END_CASE
///============================================================================================}}}
///(*==================================== Sorting station ====================================*){{{
(* Add buffer for sorting station *)
CASE eFinalResult OF
	VISION_RESULT_UNKNOWN:
		;
	VISION_RESULT_GOOD:
		Buffer_SortGood.A_Add(in := fbRotaryTable.ActualPosition + lrSortGoodDistance);
		eFinalResult 		:= VISION_RESULT_UNKNOWN;
	VISION_RESULT_CONTAMINATION_DIRTY:
		Buffer_SortDirt.A_Add(in := fbRotaryTable.ActualPosition + lrSortDirtDistance);
		eFinalResult 		:= VISION_RESULT_UNKNOWN;
	VISION_RESULT_SCRATCH_DENT:
		Buffer_SortDent.A_Add(in := fbRotaryTable.ActualPosition + lrSortDentDistance);
		eFinalResult 		:= VISION_RESULT_UNKNOWN;
	VISION_RESULT_REJECT:
		Buffer_SortReject.A_Add(in := fbRotaryTable.ActualPosition + lrSortRejectDistance);
		eFinalResult 		:= VISION_RESULT_UNKNOWN;

END_CASE
(* Shoot the product out *)
(* Good case *)
CASE uSortGoodGetPosState OF
	0://idle | check buffer
		IF Buffer_SortGood.nCount > 0 THEN
			uSortGoodGetPosState:= 10;
		END_IF
	10://get position
		Buffer_SortGood.A_Get(out => lrSortGoodPos);
		uSortGoodGetPosState := 20;
	20://waiting table move in position | command table
		bResultProcessing 	:= FALSE;
		IF LREAL_TO_INT(fbRotaryTable.ActualPosition) <= LREAL_TO_INT(lrSortGoodPos) THEN
			uSortGoodGetPosState := 30;
		END_IF
	30://shoot it
		Buffer_SortGood.A_Remove(out => lrSortGoodPos);
		doBlowGood.Out := TRUE;
		uSortGoodGetPosState := 40;
		
	40://off
		tonGoodDelay(IN := TRUE, PT := tSortValveGoodTime);
		IF tonGoodDelay.Q THEN	
			doBlowGood.Out := FALSE;
			tonGoodDelay.IN := FALSE;
			uSortGoodGetPosState := 0;
		END_IF
		
END_CASE
(* DIRT CASE *)
CASE uSortDirtGetPosState OF
	0://idle | check buffer
		IF Buffer_SortDirt.nCount > 0 THEN
			uSortDirtGetPosState:= 10;
		END_IF
	10://get position
		Buffer_SortDirt.A_Get(out => lrSortDirtPos);
		uSortDirtGetPosState := 20;
	20://waiting table move in position | command table
		bResultProcessing 	:= FALSE;
		IF LREAL_TO_INT(fbRotaryTable.ActualPosition) <= LREAL_TO_INT(lrSortDirtPos) THEN
			uSortDirtGetPosState := 30;
		END_IF
	30://shoot it
		Buffer_SortDirt.A_Remove(out => lrSortDirtPos);
		doBlowDirtScratch.Out := TRUE;
		uSortDirtGetPosState := 40;
		
	40://off
		tonDirtDelay(IN := TRUE, PT := tSortValveDirtTime);
		IF tonDirtDelay.Q THEN	
			doBlowDirtScratch.Out := FALSE;
			tonDirtDelay.IN := FALSE;
			uSortDirtGetPosState := 0;
		END_IF
		
END_CASE
(* DENT CASE *)
CASE uSortDentGetPosState OF
	0://idle | check buffer
		IF Buffer_SortDent.nCount > 0 THEN
			uSortDentGetPosState:= 10;
		END_IF
	10://get position
		Buffer_SortDent.A_Get(out => lrSortDentPos);
		uSortDentGetPosState := 20;
	20://waiting table move in position | command table
		bResultProcessing 	:= FALSE;
		IF LREAL_TO_INT(fbRotaryTable.ActualPosition) <= LREAL_TO_INT(lrSortDentPos) THEN
			uSortDentGetPosState := 30;
		END_IF
	30://shoot it
		Buffer_SortDent.A_Remove(out => lrSortDentPos);
		doBlowDentContamination.Out := TRUE;
		uSortDentGetPosState := 40;
		
	40://off
		tonDentDelay(IN := TRUE, PT := tSortValveDentTime);
		IF tonDentDelay.Q THEN	
			doBlowDentContamination.Out := FALSE;
			tonDentDelay.IN := FALSE;
			uSortDentGetPosState := 0;
		END_IF
		
END_CASE
(* REJECT CASE *)
CASE uSortRejectGetPosState OF
	0://idle | check buffer
		IF Buffer_SortReject.nCount > 0 THEN
			uSortRejectGetPosState:= 10;
		END_IF
	10://get position
		Buffer_SortReject.A_Get(out => lrSortRejectPos);
		uSortRejectGetPosState := 20;
	20://waiting table move in position | command table
		bResultProcessing 	:= FALSE;
		IF LREAL_TO_INT(fbRotaryTable.ActualPosition) <= LREAL_TO_INT(lrSortRejectPos) THEN
			uSortRejectGetPosState := 30;
		END_IF
	30://shoot it
		Buffer_SortReject.A_Remove(out => lrSortRejectPos);
		doBlowReject.Out := TRUE;
		uSortRejectGetPosState := 40;
		
	40://off
		tonRejectDelay(IN := TRUE, PT := tSortValveRejectTime);
		IF tonRejectDelay.Q THEN	
			doBlowReject.Out := FALSE;
			tonRejectDelay.IN := FALSE;
			uSortRejectGetPosState := 0;
		END_IF
		
END_CASE
///============================================================================================}}}
(* control param *)
fbRobot.ref_CR800.Override:= 5;
uBufferTableCount:= Buffer_RotaryTable.nCount;

(* Mornitoring param *)
bActive 			:= fbRotaryTable.Active;
bBusy				:= fbRotaryTable.Busy;
bError 				:= fbRotaryTable.Error;
iErrorID 			:= fbRotaryTable.ErrorID;
iAxisErrorID 		:= fbRotaryTable.ErrorID;
lrActualPosition 	:= fbRotaryTable.ActualPosition;
rActualVelocity		:= fbRotaryTable.ActualVelocity;
bPowerOn 			:= fbRotaryTable.PowerOn;
bIsHomed 			:= fbRotaryTable.IsHomed;
bInVelocity			:= fbRotaryTable.InVelocity;
bInPostion 			:= fbRotaryTable.InPosition;
bMoveActive 		:= fbRotaryTable.MoveActive;
bJogDone 			:= fbRotaryTable.JogDone;
bStopped 			:= fbRotaryTable.Stopped;
bHalted 			:= fbRotaryTable.Halted;
eStatePlcOpen		:= fbRotaryTable.StatePlcOpen;

fbRobot.ref_CR800.Override:= 30;
fbRotaryTable.Velocity 			:= 50.0;
END_METHOD

METHOD PROTECTED Production_fixing : BOOL
VAR_INST
	(* Robot *)
	RobotState 					: UINT;
	
	(* Table *)
	TableState					: UINT;
	OneStep 					: LREAL:= -30.0; //-61.1928;	(* Define by the distance between station 3 and 4 *)
	lrRelativeDistance 			: LREAL;
	bProductAboveTable 			: BOOL;				(* Signal Robot is at the table *)
	bGetPictureStation3			: BOOL; 			(* Cmd get picture st3 to vision system *)
	bGetPictureStation4 		: BOOL; 			(* Cmd get picture st4 to vision system *)
	bResultProcessing 			: BOOL;				(* Request result from vision system, then add buffer for sorting station *)
	
	(* Buffer *)
	BufferState : UINT;
	Buffer_RotaryTable			: FB_DataSetFifo_1; 	(* Contain the position of all product on the table *)
	Buffer_Station3				: FB_DataSetFifo_1;	(* Contain the trigger position *)
	Buffer_Station4				: FB_DataSetFifo_1;	(* Contain the trigger position *)
	
	(* Sorting Station *)
	Buffer_SortGood				: FB_DataSetFifo_1;
	Buffer_SortDirt				: FB_DataSetFifo_1;
	Buffer_SortDent				: FB_DataSetFifo_1;
	Buffer_SortReject			: FB_DataSetFifo_1;
	
	
	
	lrSortGoodPos				: LREAL;
	lrSortDirtPos				: LREAL;
	lrSortDentPos				: LREAL;
	lrSortRejectPos				: LREAL;
	
	uSortGoodGetPosState		: UINT; 			(* state machine of get sort position from buffer *)
	uSortDirtGetPosState		: UINT;
	uSortDentGetPosState		: UINT;
	uSortRejectGetPosState		: UINT;
		
	tonGoodDelay				: TON;				(* one shoot of good delay valve *)
	tonDirtDelay				: TON;				(* one shoot of dirt delay valve *)
	tonDentDelay				: TON;				(* one shoot of dent delay valve *)								
	tonRejectDelay				: TON;				(* one shoot of reject delay valve *)	
							

	
	(*=== Vision ===*)
	Vision3State 		: UINT;
	Vision4State		: UINT;
	lrCapPosStation3 	: LREAL;
	lrCapPosStation4	: LREAL;
	bGood 				: BOOL;
	bAtVision3 			: BOOL;	(* Product is at vision 3 *)
	bAtVision4 			: BOOL;	(* Product is at vision 4 *)
	eFinalResult		: E_VisionResult;

	(* Axis status flags *)
	bActive					: BOOL;
	bBusy					: BOOL;								(* Function block currently executes one of the requests *)
	bError					: BOOL;								(* Error status flag *)
	iErrorID				: UDINT;							(* Error ID *)
	iAxisErrorID			: UDINT;							(* Axis error ID*)
	lrActualPosition		: LREAL;							(* Actual axis position in selected units *)
	rActualVelocity			: REAL;								(* Actual axis velocity in selected units *)
	bPowerOn 				: BOOL;								(* Power On status bit *)
	bIsHomed				: BOOL;								(* Axis has been homed even once *)
	bInVelocity				: BOOL;								(* Axis is moving in target velocity *)
	bInPostion				: BOOL;								(* Axis reached target position *)
	bMoveActive				: BOOL;								(* Axis is moving to target position *)
	bJogDone				: BOOL;								(* Axis manual movement by jog done *)
	bStopped				: BOOL;								(* Axis movement has been stopped *)
	bHalted					: BOOL;								(* Axis movement has been halted *)
	eStatePlcOpen			: E_AxisStatePlcOpen;
	
	uBufferTableCount : UDINT;
	
	(* testing bit *)
	bResultTest : BOOL;
	bResultGood : BOOL;
	bResultDirt : BOOL;
	bResultDent : BOOL;
	bResultReject : BOOL;

	(**)
	iTableSupervisor 	: UINT;
	iTableExecutor 		: UINT;
	
	Buffer_Sorting		: FB_DataSetFifo_1;	(* Contain the trigger position *)
	
	lrStation3Location : LREAL;
	lrStation4Location : LREAL;
	lrStationSortLocation : LREAL;
	lrTargetLocation : LREAL;
	
	bBufferTest : BOOL;
	
END_VAR
///(*==================================== Robot + Vision process ====================================*){{{
CASE RobotState OF	
	0://IDLE go bowl
		fbRobot.MR_GoBowl();
		IF NOT fbRobot.Busy THEN
			RobotState := 5;
		END_IF		
	5://product detected
		IF diProductPresenceBowl.In THEN (* waiting product *)
			RobotState := 6;
		END_IF
	
	6://go input
		fbRobot.MR_GoInputProduct();
		IF NOT fbRobot.Busy THEN
			RobotState := 7;
		END_IF
		
	7://robot pick
		fbRobot.MR_Pick();
		IF NOT fbRobot.Busy THEN
			RobotState := 10;
		END_IF 
		
	10://go to station 1
		fbRobot.MR_GoStation1();
		IF NOT fbRobot.Busy THEN
			RobotState := 20;
		END_IF
		
	20://double trig cam 1+2
		IF doTriggerCam1.Command(PulseWidth:=T#1MS, DelayTimeForSecondTrigger := T#35MS) AND
			doTriggerCam2.Command(PulseWidth:=T#1MS, DelayTimeForSecondTrigger := T#35MS) THEN
			RobotState:= 30;
		END_IF
	30://go to station 2
		fbRobot.MR_GoStation2();
		IF NOT fbRobot.Busy THEN
			RobotState := 40;
		END_IF
	40://double trig cam 3+4
		IF doTriggerCam3.Command(PulseWidth:=T#1MS, DelayTimeForSecondTrigger := T#35MS) AND
			doTriggerCam4.Command(PulseWidth:=T#1MS, DelayTimeForSecondTrigger := T#35MS) THEN
			RobotState := 50;
		END_IF
	50://goto rotary table
		fbRobot.MR_GoRotaryTable();
		IF NOT fbRobot.Busy THEN
			bProductAboveTable := TRUE;		
			RobotState:= 60;
		END_IF
	60://waiting command from table
		;
		
END_CASE
///============================================================================================}}}
(* TABLE SUPERVISOR *)
CASE iTableSupervisor OF
	0:
		IF bProductAboveTable THEN			
			IF iTableExecutor = 0 THEN//IDLE
				RobotState:=60;
			END_IF
		END_IF
		
END_CASE
(* TABLE EXECUTOR *)
CASE iTableExecutor OF
	0: //IDLE
		;
	10://TAKE PRODUCT
		
	20://ADD BUFFER
		Buffer_Station3.A_Add(in:= fbRotaryTable.ActualPosition + 2*OneStep); 	(* station position *)
		Buffer_Station4.A_Add(in:= fbRotaryTable.ActualPosition + 4*OneStep);	(* station position *)
		
		Buffer_RotaryTable.A_Add(in:= fbRotaryTable.ActualPosition + OneStep);	(* place position *)
		Buffer_RotaryTable.A_Add(in:= fbRotaryTable.ActualPosition + OneStep);	(* place position *)
		Buffer_RotaryTable.A_Add(in:= fbRotaryTable.ActualPosition + OneStep);	(* place position *)
		Buffer_RotaryTable.A_Add(in:= fbRotaryTable.ActualPosition + OneStep);	(* place position *)
		
		iTableExecutor := 30;
	30://calc the position
		IF Buffer_Station3.nCount > 0 AND Buffer_Station4.nCount > 0 THEN
			Buffer_Station3.A_Get(out => lrStation3Location);
			Buffer_Station4.A_Get(out => lrStation4Location);
			
			IF LREAL_TO_LINT(lrStation3Location) > LREAL_TO_LINT(lrStation4Location) THEN
				lrTargetLocation := lrStation3Location;
				Buffer_Station3.A_Remove(out => lrStation3Location);
				
			ELSIF LREAL_TO_LINT(lrStation3Location) < LREAL_TO_LINT(lrStation4Location) THEN
				lrTargetLocation := lrStation4Location;
				Buffer_Station4.A_Remove(out => lrStation4Location);
				
			ELSE
				lrTargetLocation := lrStation3Location;
				Buffer_Station3.A_Remove(out => lrStation3Location);
				Buffer_Station4.A_Remove(out => lrStation4Location);
			
			END_IF
			iTableExecutor := 40;
			
		ELSIF Buffer_Station3.nCount = 0 AND Buffer_Station4.nCount = 0 THEN
			iTableExecutor := 0;//IDLE
			
		ELSE
			IF Buffer_Station3.nCount = 0 THEN
				lrTargetLocation := lrStation4Location;
				Buffer_Station4.A_Remove(out => lrStation4Location);
				
			ELSE
				lrTargetLocation := lrStation3Location;
				Buffer_Station3.A_Remove(out => lrStation3Location);
				
			END_IF
			iTableExecutor := 40;
		END_IF
		
	40://
		fbRotaryTable.MR_MoveAbsolute(lrAbsolutePosition := lrTargetLocation);
		IF fbRotaryTable.InPosition THEN
			iTableExecutor := 30;
		END_IF
		
		
END_CASE
///============================================================================================}}}
(* control param *)
fbRobot.ref_CR800.Override:= 5;
uBufferTableCount:= Buffer_RotaryTable.nCount;

(* Mornitoring param *)
bActive 			:= fbRotaryTable.Active;
bBusy				:= fbRotaryTable.Busy;
bError 				:= fbRotaryTable.Error;
iErrorID 			:= fbRotaryTable.ErrorID;
iAxisErrorID 		:= fbRotaryTable.ErrorID;
lrActualPosition 	:= fbRotaryTable.ActualPosition;
rActualVelocity		:= fbRotaryTable.ActualVelocity;
bPowerOn 			:= fbRotaryTable.PowerOn;
bIsHomed 			:= fbRotaryTable.IsHomed;
bInVelocity			:= fbRotaryTable.InVelocity;
bInPostion 			:= fbRotaryTable.InPosition;
bMoveActive 		:= fbRotaryTable.MoveActive;
bJogDone 			:= fbRotaryTable.JogDone;
bStopped 			:= fbRotaryTable.Stopped;
bHalted 			:= fbRotaryTable.Halted;
eStatePlcOpen		:= fbRotaryTable.StatePlcOpen;

fbRobot.ref_CR800.Override:= 30;
fbRotaryTable.Velocity 			:= 50.0;
END_METHOD

METHOD PROTECTED Robot_Process
VAR_INST
	(* Equipment module sequences *)
	RobotState : UINT;
	
END_VAR
CASE RobotState OF	
	0://IDLE go bowl
		fbRobot.MR_GoBowl();
		IF NOT fbRobot.Busy THEN
			RobotState := 5;
		END_IF		
	5://product detected
		IF diProductPresenceBowl.In THEN (* waiting product *)
			RobotState := 6;
		END_IF
	
	6://go input
		fbRobot.MR_GoInputProduct();
		IF NOT fbRobot.Busy THEN
			RobotState := 7;
		END_IF
		
	7://robot pick
		fbRobot.MR_Pick();
		IF NOT fbRobot.Busy THEN
			RobotState := 10;
		END_IF 
		
	10://go to station 1
		fbRobot.MR_GoStation1();
		IF NOT fbRobot.Busy THEN
			RobotState := 20;
		END_IF
		
	20://double trig cam 1+2
		IF doTriggerCam1.Command(PulseWidth:=T#1MS, DelayTimeForSecondTrigger := T#35MS) AND
			doTriggerCam2.Command(PulseWidth:=T#1MS, DelayTimeForSecondTrigger := T#35MS) THEN
			RobotState:= 30;
		END_IF
	30://go to station 2
		fbRobot.MR_GoStation2();
		IF NOT fbRobot.Busy THEN
			RobotState := 40;
		END_IF
	40://double trig cam 3+4
		IF doTriggerCam3.Command(PulseWidth:=T#1MS, DelayTimeForSecondTrigger := T#35MS) AND
			doTriggerCam4.Command(PulseWidth:=T#1MS, DelayTimeForSecondTrigger := T#35MS) THEN
			RobotState := 50;
		END_IF
	50://goto rotary table
		fbRobot.MR_GoRotaryTable();
		IF NOT fbRobot.Busy THEN
			//bProductAboveTable := TRUE;		
			RobotState:= 60;
		END_IF
	60://waiting command from table
		fbRobot.MR_Place();
		IF NOT fbRobot.Busy THEN
			RobotState := 0;
		END_IF
		
END_CASE
END_METHOD

METHOD robotcamtest : BOOL
VAR_INST
	RobotProcess:UINT;
END_VAR
fbRobot.ref_CR800.Override:= 5;
CASE RobotProcess OF
	
	0://IDLE go bowl
		fbRobot.MR_GoBowl();
		IF NOT fbRobot.Busy THEN
			RobotProcess := 5;
		END_IF		
	5://product detected
		IF diProductPresenceBowl.In THEN (* waiting product *)
			RobotProcess := 6;
		END_IF
	
	6://go input
		fbRobot.MR_GoInputProduct();
		IF NOT fbRobot.Busy THEN
			RobotProcess := 7;
		END_IF
		
	7://robot pick
		fbRobot.MR_Pick();
		IF NOT fbRobot.Busy THEN
			RobotProcess := 10;
		END_IF 
		
	10://go to station 1
		fbRobot.MR_GoStation1();
		IF NOT fbRobot.Busy THEN
			RobotProcess := 20;
		END_IF
END_CASE
END_METHOD

PROPERTY Robots : REFERENCE TO FB_Robot
GET
Robots REF= fbRobot;
END_GET
END_PROPERTY

PROPERTY StateInit : REFERENCE TO E_MachineCtrlStateInit
GET
StateInit REF= eMachineStateInit;
END_GET
END_PROPERTY

PROPERTY StateUninitialized : REFERENCE TO E_MachineCtrlStateUninitialized
GET
StateUninitialized REF= eMachineStateUninitialized;
END_GET
END_PROPERTY

METHOD TableProcess : BOOL
VAR_INST
	(*=== Table ===*)
	TableState : UINT;
	OneStep : LREAL:= -61.1928;
	lrRelativeDistance : LREAL;
	
	(* Axis status flags *)
	bActive					: BOOL;
	bBusy					: BOOL;								(* Function block currently executes one of the requests *)
	bError					: BOOL;								(* Error status flag *)
	iErrorID				: UDINT;							(* Error ID *)
	iAxisErrorID			: UDINT;							(* Axis error ID*)
	lrActualPosition		: LREAL;							(* Actual axis position in selected units *)
	rActualVelocity			: REAL;								(* Actual axis velocity in selected units *)
	bPowerOn 				: BOOL;								(* Power On status bit *)
	bIsHomed				: BOOL;								(* Axis has been homed even once *)
	bInVelocity				: BOOL;								(* Axis is moving in target velocity *)
	bInPostion				: BOOL;								(* Axis reached target position *)
	bMoveActive				: BOOL;								(* Axis is moving to target position *)
	bJogDone				: BOOL;								(* Axis manual movement by jog done *)
	bStopped				: BOOL;								(* Axis movement has been stopped *)
	bHalted					: BOOL;								(* Axis movement has been halted *)
	eStatePlcOpen			: E_AxisStatePlcOpen;				(* Current PLCOpen state of axis *)
	
	
	(* Buffer *)
	Buffer_RotaryTable			: FB_DataSetFifo; 	(* Contain the position of all product on the table *)
	Buffer_Station3				: FB_DataSetFifo;	(* Contain the trigger position *)
	Buffer_Station4				: FB_DataSetFifo;	(* Contain the trigger position *)
	
	(*=== Vision ===*)
	Vision3State : UINT;
	Vision4State: UINT;
	lrCapPosStation3 : LREAL;
	lrCapPosStation4: LREAL;
	//lrActualPosition :LREAL;
	bBufferReset : BOOL;
END_VAR
CASE TableState OF
	0://product in
		IF diProductPresenceBowl.In THEN (* waiting product *)
			TableState := 10;
		END_IF
	10://buffer table, station 3, station 4
		IF Buffer_RotaryTable.Add2Data(in1 := OneStep, in2 := OneStep) THEN
			IF Buffer_Station3.Add1Data(in := fbRotaryTable.ActualPosition + OneStep) THEN
				IF Buffer_Station4.Add1Data(in := fbRotaryTable.ActualPosition + 2*OneStep) THEN
					TableState := 20;
		
				END_IF				
			END_IF
		END_IF
	20://take distance
		Buffer_RotaryTable.Remove(out => lrRelativeDistance);
		IF Buffer_RotaryTable.OK THEN
			TableState := 30;
		END_IF
	30://move distance
		fbRotaryTable.MR_MoveRelative(lrRelativeDistance);
		IF fbRotaryTable.InPosition THEN
			TableState := 40;
		END_IF
	40://check
		IF Buffer_RotaryTable.Count >0 THEN
			TableState := 20;
		ELSE 
			TableState := 0;
		END_IF
END_CASE

lrActualPosition := fbRotaryTable.ActualPosition;

CASE Vision3State OF
	0://take capture position
		Buffer_Station3.Remove(out => lrCapPosStation3);
		IF Buffer_Station3.OK THEN
			Vision3State := 10;
		END_IF
	10://waiting table move in pos
		IF LREAL_TO_INT(fbRotaryTable.ActualPosition) = LREAL_TO_INT(lrCapPosStation3) THEN
			Vision3State:= 20;
			
		END_IF
	20://capture
		IF fbRTCVision.M_CommandStation3(PulseWidth:= T#1MS, DelayTimeForSecondTrigger:= T#33MS) THEN
			Vision3State:= 0;
		END_IF

END_CASE

CASE Vision4State OF
	0://take capture position
		Buffer_Station4.Remove(out => lrCapPosStation4);
		IF Buffer_Station4.OK THEN
			Vision4State := 10;
		END_IF
	10://waiting table move in pos
		IF LREAL_TO_INT(fbRotaryTable.ActualPosition) = LREAL_TO_INT(lrCapPosStation4) THEN
			Vision4State:= 20;
			
		END_IF
	20://capture
		IF fbRTCVision.M_CommandStation4(PulseWidth:= T#1MS, DelayTimeForSecondTrigger:= T#33MS) THEN
			Vision4State:= 0;
		END_IF

END_CASE
(*===== Utilities =====*)
IF bBufferReset THEN
	Buffer_Station3.Reset();
	Buffer_Station4.Reset();
	Buffer_RotaryTable.Reset();
//	IF Buffer_Station3.OK AND Buffer_Station4.OK AND Buffer_RotaryTable.OK THEN
		
//	END_IF
END_IF

bActive 			:= fbRotaryTable.Active;
bBusy				:= fbRotaryTable.Busy;
bError 				:= fbRotaryTable.Error;
iErrorID 			:= fbRotaryTable.ErrorID;
iAxisErrorID 		:= fbRotaryTable.ErrorID;
lrActualPosition 	:= fbRotaryTable.ActualPosition;
rActualVelocity		:= fbRotaryTable.ActualVelocity;
bPowerOn 			:= fbRotaryTable.PowerOn;
bIsHomed 			:= fbRotaryTable.IsHomed;
bInVelocity			:= fbRotaryTable.InVelocity;
bInPostion 			:= fbRotaryTable.InPosition;
bMoveActive 		:= fbRotaryTable.MoveActive;
bJogDone 			:= fbRotaryTable.JogDone;
bStopped 			:= fbRotaryTable.Stopped;
bHalted 			:= fbRotaryTable.Halted;
eStatePlcOpen		:= fbRotaryTable.StatePlcOpen;
END_METHOD

METHOD tableRefer : BOOL
VAR_INST
	bparamhome : BOOL;
	bFirstCycle 	: BOOL;
	
	stLiftHomingOptions				: ST_HomingOptions; 

	
	bInit					: BOOL;								(* Power on axis and prepare to work *)
	bAbort					: BOOL;								(* Power off axis and reset status flags *)
	bHome					: BOOL;								(* Home to reference point *)
	bMoveVelocity			: BOOL;								(* Start motion with constant velocity *)
	bMoveAbsolute			: BOOL;								(* Move to absolute position *)
	bMoveAdditive			: BOOL;								(* Move by distance *)
	bMoveRelative			: BOOL;								(* Move by distance *)
	bJog					: BOOL;								(* Start manual jog movement *)
	bStop					: BOOL;								(* High priority stop command *)
	bHalt					: BOOL;								(* Halt current motion, next motion command will abort this command *)
	bReset					: BOOL;								(* Reset axis and return to READY state *)
	
	(* General parameters *)
	bModulo					: BOOL := FALSE;					(* Axis is periodic *)
	lrOverride				: LREAL;							(* Axis velocity override in percents [%] *)
	lrVelocity 				: LREAL;							(* Axis velocirt in measurement units per second *)
	lrAcceleration			: LREAL;							(* Axis acceleration in measurement units per sercond^2 *)
	lrDeceleration 			: LREAL;							(* Axis deceleration in measurement units per sercond^2 *)
	lrJerk					: LREAL;							(* Axis jerk in measurement unit per sercond^3 *)
	lrAbsolutePosition		: LREAL;							(* Target position for MC_MoveAbsolute function *)
	lrRelativeDistance		: LREAL;							(* Relative distance to move for MC_MoveRelative/Additive fuctions *)
	lrHomePosition			: LREAL;							(* This parameters is used to set axis position while performing homing procedure *)
	
	(* Jog function parameters *)	
	lrJogPosition			: LREAL;							(* Relative position to move for jog feature *)
	lrJogVelocity			: LREAL;							(* Jog movement velocity *)
	lrJogAcceleration		: LREAL;							(* Jog movement acceleration *)
	lrJogDeceleration		: LREAL;							(* Jog movement deceleration *)
	lrJogJerk				: LREAL;							(* Jog movement jerk *)
	eJogMode				: E_JogMode;						(* Jog movement mode *)
	eJogDirection			: E_AxisJogDirection;				(* Direction of jog movement *)
	
	(* Stop function parameters *)
	lrStopDeceleration		: LREAL;							(* Stop deceleration *)
	lrStopJerk 				: LREAL;							(* Stop jerk *)
	
	(* Other parameters *)
	stOptions				: ST_MoveOptions;					(* Additional movement options *)
	eDirection				: Tc2_MC2.MC_Direction;				(* Axis movement direction for MC_MoveVelocity *)
	eBufferMode 			: MC_BufferMode := MC_Aborting;		(* Axis buffering mode *)
	
	(* Axis status flags *)
	bActive					: BOOL;
	bBusy					: BOOL;								(* Function block currently executes one of the requests *)
	bError					: BOOL;								(* Error status flag *)
	iErrorID				: UDINT;							(* Error ID *)
	iAxisErrorID			: UDINT;							(* Axis error ID*)
	lrActualPosition		: LREAL;							(* Actual axis position in selected units *)
	rActualVelocity			: REAL;								(* Actual axis velocity in selected units *)
	bPowerOn 				: BOOL;								(* Power On status bit *)
	bIsHomed				: BOOL;								(* Axis has been homed even once *)
	bInVelocity				: BOOL;								(* Axis is moving in target velocity *)
	bInPostion				: BOOL;								(* Axis reached target position *)
	bMoveActive				: BOOL;								(* Axis is moving to target position *)
	bJogDone				: BOOL;								(* Axis manual movement by jog done *)
	bStopped				: BOOL;								(* Axis movement has been stopped *)
	bHalted					: BOOL;								(* Axis movement has been halted *)
	eStatePlcOpen			: E_AxisStatePlcOpen;				(* Current PLCOpen state of axis *)
	
	iAxisStateMachine		: INT;
END_VAR
IF bFirstCycle THEN
	
	lrOverride 			:= 100.0;
	lrVelocity 			:= 100.0;
	lrAcceleration		:= 1500.0;
	lrDeceleration		:= 1500.0;
	lrJerk				:= 1500.0;
	lrAbsolutePosition	:= 0.0;
	lrRelativeDistance	:= 0.0;
	lrHomePosition		:= 0.0;
	
	lrJogPosition		:= 0.0;
	lrJogVelocity 		:= 25.0;
	lrJogAcceleration	:= 250.0;
	lrJogDeceleration	:= 250.0;
	lrJogJerk			:= 250.0;
	
	lrStopDeceleration	:= 250.0;
	lrStopJerk			:= 250.0;	
	
	fbRotaryTable.Override			:= lrOverride;
	fbRotaryTable.Velocity 		:= lrVelocity;
	fbRotaryTable.Acceleration 	:= lrAcceleration;
	fbRotaryTable.Deceleration 	:= lrDeceleration;
	fbRotaryTable.Jerk 			:= lrJerk;
	fbRotaryTable.JogMode			:= eJogMode;
	fbRotaryTable.JogDirection		:= eJogDirection;
	fbRotaryTable.JogVelocity 		:= lrJogVelocity;
	fbRotaryTable.JogAcceleration 	:= lrJogAcceleration;
	fbRotaryTable.JogDeceleration 	:= lrJogDeceleration;
	fbRotaryTable.JogJerk 			:= lrJogJerk;
	fbRotaryTable.StopDeceleration := lrStopDeceleration;
	fbRotaryTable.StopJerk 		:= lrStopJerk;
END_IF

IF bparamhome THEN
	bparamhome := FALSE;
	
	fbRotaryTable.MR_FirstCycle(	sName				:= CONCAT(STR1 := '', STR2 := CONCAT(STR1 := ':', STR2 := '')),
							sMeasurementUnits 	:= '',
							bModulo				:= FALSE);
								
	stLiftHomingOptions.SearchDirection := Tc2_MC2.MC_Direction.MC_Negative_Direction;
	stLiftHomingOptions.SearchVelocity 	:= 50.0;
	stLiftHomingOptions.SyncDirection 	:= Tc2_MC2.MC_Direction.MC_Positive_Direction;
	stLiftHomingOptions.SyncVelocity	:= 10.0;
	
	fbRotaryTable.Override 		:= 100.0;
	fbRotaryTable.Velocity 		:= 50.0;
	fbRotaryTable.Acceleration 	:= 150.0;
	fbRotaryTable.Deceleration 	:= 150.0;
	fbRotaryTable.Jerk 			:= 1500.0;
	fbRotaryTable.HomingMode		:= MC_HomingMode.MC_DefaultHoming;
	fbRotaryTable.HomingOptions 	:= stLiftHomingOptions;
	fbRotaryTable.JogPosition 		:= 0.0;
	fbRotaryTable.JogVelocity 		:= 40.0;
	fbRotaryTable.JogAcceleration 	:= 100.0;
	fbRotaryTable.JogDeceleration 	:= 100.0;
	fbRotaryTable.JogJerk 			:= 1000.0;
	fbRotaryTable.StopDeceleration	:= 100.0;
	fbRotaryTable.StopJerk 		:= 1000.0;

	
END_IF

bActive 			:= fbRotaryTable.Active;
bBusy				:= fbRotaryTable.Busy;
bError 				:= fbRotaryTable.Error;
iErrorID 			:= fbRotaryTable.ErrorID;
iAxisErrorID 		:= fbRotaryTable.ErrorID;
lrActualPosition 	:= fbRotaryTable.ActualPosition;
rActualVelocity		:= fbRotaryTable.ActualVelocity;
bPowerOn 			:= fbRotaryTable.PowerOn;
bIsHomed 			:= fbRotaryTable.IsHomed;
bInVelocity			:= fbRotaryTable.InVelocity;
bInPostion 			:= fbRotaryTable.InPosition;
bMoveActive 		:= fbRotaryTable.MoveActive;
bJogDone 			:= fbRotaryTable.JogDone;
bStopped 			:= fbRotaryTable.Stopped;
bHalted 			:= fbRotaryTable.Halted;
eStatePlcOpen		:= fbRotaryTable.StatePlcOpen;

IF bStop THEN
	bStop := FALSE;
	iAxisStateMachine := 20;
	
ELSIF bHalt THEN
	bHalt := FALSE;
	iAxisStateMachine := 30;
	
ELSIF bReset THEN
	bReset := FALSE;
	iAxisStateMachine := 40;
	
ELSIF bAbort THEN
	bAbort := FALSE;
	iAxisStateMachine := 110;
	
END_IF

CASE iAxisStateMachine OF
	(* Starts seqence *)
	0:
		IF bInit THEN
			bInit := FALSE;
			iAxisStateMachine := 10;

		ELSIF bHome THEN
			bHome := FALSE;
			iAxisStateMachine := 50;
			
		ELSIF bMoveVelocity THEN
			bMoveVelocity := FALSE;
			iAxisStateMachine := 60;
		
		ELSIF bMoveAbsolute THEN
			bMoveAbsolute := FALSE;
			iAxisStateMachine := 70;
		
		ELSIF bMoveAdditive THEN
			bMoveAdditive := FALSE;
			iAxisStateMachine := 80;
			
		ELSIF bMoveRelative THEN
			bMoveRelative := FALSE;
			iAxisStateMachine := 90;
			
		ELSIF bJog THEN
			iAxisStateMachine := 100;
		
		END_IF
		
	(* Initialization *)
	10:
		fbRotaryTable.MR_Init();	
		IF fbRotaryTable.PowerOn THEN
			iAxisStateMachine := 0;
		END_IF
		
	(* Stopping *)
	20:
		bJog := FALSE;
		bMoveAbsolute := FALSE;
		bMoveAdditive := FALSE;
		bMoveRelative := FALSE;
		bMoveVelocity := FALSE;
		
		IF fbRotaryTable.MR_Stop() THEN
			iAxisStateMachine := 0;
		END_IF
		
	(* Halting *)
	30:
		bJog := FALSE;
		bMoveAbsolute := FALSE;
		bMoveAdditive := FALSE;
		bMoveRelative := FALSE;
		bMoveVelocity := FALSE;
		
		fbRotaryTable.MR_Halt();
		IF fbRotaryTable.Halted THEN
			iAxisStateMachine := 0;
		END_IF
		
	(* Resetting *)
	40:
		fbRotaryTable.MR_Reset(); 
		IF NOT fbRotaryTable.Error THEN
			iAxisStateMachine := 0;
		END_IF
	
	(* Homing *)
	50: 
		fbRotaryTable.MR_Home(lrHomePosition:=-2.5);
		IF fbRotaryTable.IsHomed THEN	
			iAxisStateMachine := 0;
		END_IF
	
	(* Move velocity *)	
	60: 
		fbRotaryTable.MR_MoveVelocity();
		IF fbRotaryTable.InVelocity THEN
			iAxisStateMachine := 0;
		END_IF
		
	(* Move absolute *)
	70: 
		fbRotaryTable.MR_MoveAbsolute(lrAbsolutePosition);
		IF fbRotaryTable.InPosition THEN
			iAxisStateMachine := 0;
		END_IF
		
	(* Move additive *)	
	80: 
		fbRotaryTable.MR_MoveAdditive(lrRelativeDistance);
		IF fbRotaryTable.InPosition THEN
			iAxisStateMachine := 0;
		END_IF
		
	(* Move relative *)	
	90: 
		fbRotaryTable.MR_MoveRelative(lrRelativeDistance);
		IF fbRotaryTable.InPosition THEN
			iAxisStateMachine := 0;
		END_IF
		
	(* Jog movement *)	
	100: 
		fbRotaryTable.MR_Jog(bJog);
		IF fbRotaryTable.JogDone THEN
			bJog := FALSE;
			iAxisStateMachine := 0;
		END_IF
		
	(* Deinitialization *)	
	110: 
		fbRotaryTable.MR_Abort();
		IF NOT fbRotaryTable.PowerOn THEN
			iAxisStateMachine := 0;
		END_IF		
END_CASE
END_METHOD

METHOD Test : BOOL
VAR_INST
	(* Robot *)
	RobotState 					: UINT;
	
	(* Table *)
	TableState					: UINT;
	OneStep 					: LREAL:= -60.0; //-61.1928;	(* Define by the distance between station 3 and 4 *)
	lrRelativeDistance 			: LREAL;
	bProductAboveTable 			: BOOL;				(* Signal Robot is at the table *)
	bGetPictureStation3			: BOOL; 			(* Cmd get picture st3 to vision system *)
	bGetPictureStation4 		: BOOL; 			(* Cmd get picture st4 to vision system *)
	bResultProcessing 			: BOOL;				(* Request result from vision system, then add buffer for sorting station *)
	
	(* Buffer *)
	BufferState : UINT;
	Buffer_RotaryTable			: FB_DataSetFifo_1; 	(* Contain the position of all product on the table *)
	Buffer_Station3				: FB_DataSetFifo_1;	(* Contain the trigger position *)
	Buffer_Station4				: FB_DataSetFifo_1;	(* Contain the trigger position *)
	
	(* Sorting Station *)
	Buffer_SortGood				: FB_DataSetFifo_1;
	Buffer_SortDirt				: FB_DataSetFifo_1;
	Buffer_SortDent				: FB_DataSetFifo_1;
	Buffer_SortReject			: FB_DataSetFifo_1;
	
	
	
	lrSortGoodPos				: LREAL;
	lrSortDirtPos				: LREAL;
	lrSortDentPos				: LREAL;
	lrSortRejectPos				: LREAL;
	
	uSortGoodGetPosState		: UINT; 			(* state machine of get sort position from buffer *)
	uSortDirtGetPosState		: UINT;
	uSortDentGetPosState		: UINT;
	uSortRejectGetPosState		: UINT;
		
	tonGoodDelay				: TON;				(* one shoot of good delay valve *)
	tonDirtDelay				: TON;				(* one shoot of dirt delay valve *)
	tonDentDelay				: TON;				(* one shoot of dent delay valve *)								
	tonRejectDelay				: TON;				(* one shoot of reject delay valve *)	
							

	
	(*=== Vision ===*)
	Vision3State 		: UINT;
	Vision4State		: UINT;
	lrCapPosStation3 	: LREAL;
	lrCapPosStation4	: LREAL;
	bGood 				: BOOL;
	bAtVision3 			: BOOL;	(* Product is at vision 3 *)
	bAtVision4 			: BOOL;	(* Product is at vision 4 *)
	eFinalResult		: E_VisionResult;

	(* Axis status flags *)
	bActive					: BOOL;
	bBusy					: BOOL;								(* Function block currently executes one of the requests *)
	bError					: BOOL;								(* Error status flag *)
	iErrorID				: UDINT;							(* Error ID *)
	iAxisErrorID			: UDINT;							(* Axis error ID*)
	lrActualPosition		: LREAL;							(* Actual axis position in selected units *)
	rActualVelocity			: REAL;								(* Actual axis velocity in selected units *)
	bPowerOn 				: BOOL;								(* Power On status bit *)
	bIsHomed				: BOOL;								(* Axis has been homed even once *)
	bInVelocity				: BOOL;								(* Axis is moving in target velocity *)
	bInPostion				: BOOL;								(* Axis reached target position *)
	bMoveActive				: BOOL;								(* Axis is moving to target position *)
	bJogDone				: BOOL;								(* Axis manual movement by jog done *)
	bStopped				: BOOL;								(* Axis movement has been stopped *)
	bHalted					: BOOL;								(* Axis movement has been halted *)
	eStatePlcOpen			: E_AxisStatePlcOpen;
	
	uBufferTableCount : UDINT;
	
	(* testing bit *)
	bResultTest : BOOL;
	bResultGood : BOOL;
	bResultDirt : BOOL;
	bResultDent : BOOL;
	bResultReject : BOOL;

	lrStation3Location : LREAL;
	lrStation4Location : LREAL;
	lrTargetLocation : LREAL;
	
END_VAR
///(*==================================== Robot + Vision process ====================================*){{{
CASE RobotState OF	
	0://IDLE go bowl
		fbRobot.MR_GoBowl();
		IF NOT fbRobot.Busy THEN
			RobotState := 5;
		END_IF		
	5://product detected
		IF diProductPresenceBowl.In THEN (* waiting product *)
			RobotState := 6;
		END_IF
	
	6://go input
		fbRobot.MR_GoInputProduct();
		IF NOT fbRobot.Busy THEN
			RobotState := 7;
		END_IF
		
	7://robot pick
		fbRobot.MR_Pick();
		IF NOT fbRobot.Busy THEN
			RobotState := 10;
		END_IF 
		
	10://go to station 1
		fbRobot.MR_GoStation1();
		IF NOT fbRobot.Busy THEN
			RobotState := 20;
		END_IF
		
	20://double trig cam 1+2
		IF doTriggerCam1.Command(PulseWidth:=T#1MS, DelayTimeForSecondTrigger := T#35MS) AND
			doTriggerCam2.Command(PulseWidth:=T#1MS, DelayTimeForSecondTrigger := T#35MS) THEN
			RobotState:= 30;
		END_IF
	30://go to station 2
		fbRobot.MR_GoStation2();
		IF NOT fbRobot.Busy THEN
			RobotState := 40;
		END_IF
	40://double trig cam 3+4
		IF doTriggerCam3.Command(PulseWidth:=T#1MS, DelayTimeForSecondTrigger := T#35MS) AND
			doTriggerCam4.Command(PulseWidth:=T#1MS, DelayTimeForSecondTrigger := T#35MS) THEN
			RobotState := 50;
		END_IF
	50://goto rotary table
		fbRobot.MR_GoRotaryTable();
		IF NOT fbRobot.Busy THEN
			bProductAboveTable := TRUE;		
			RobotState:= 60;
		END_IF
	60://waiting command from table
		;
		
END_CASE
///============================================================================================}}}
///(*==================================== Table process ====================================*){{{
CASE TableState OF
	0:// idle | waiting for product
		IF bProductAboveTable THEN
			TableState:= 10;
		END_IF
	10://command place product and reset robot sequence
		fbRobot.MR_Place();
		IF NOT fbRobot.Busy THEN
			bProductAboveTable := FALSE;
			RobotState := 0;
			TableState := 20;
		END_IF
	20://add buffer for st 3+4, table
		Buffer_Station3.A_Add(in:= fbRotaryTable.ActualPosition + 2*OneStep); 	(* station position *)
		Buffer_Station4.A_Add(in:= fbRotaryTable.ActualPosition + 4*OneStep);	(* station position *)
		
		Buffer_RotaryTable.A_Add(in:= fbRotaryTable.ActualPosition + OneStep);	(* place position *)
		Buffer_RotaryTable.A_Add(in:= fbRotaryTable.ActualPosition + OneStep);	(* place position *)
		Buffer_RotaryTable.A_Add(in:= fbRotaryTable.ActualPosition + OneStep);	(* place position *)
		Buffer_RotaryTable.A_Add(in:= fbRotaryTable.ActualPosition + OneStep);	(* place position *)
		TableState := 25;
		
	25://CALC POSITION
		IF Buffer_Station3.nCount > 0 AND Buffer_Station4.nCount > 0 THEN
			Buffer_Station3.A_Get(out => lrStation3Location);
			Buffer_Station4.A_Get(out => lrStation4Location);
			
			IF LREAL_TO_LINT(lrStation3Location) > LREAL_TO_LINT(lrStation4Location) THEN
				lrTargetLocation := lrStation3Location;
				Buffer_Station3.A_Remove(out => lrStation3Location);
				
			ELSIF LREAL_TO_LINT(lrStation3Location) < LREAL_TO_LINT(lrStation4Location) THEN
				lrTargetLocation := lrStation4Location;
				Buffer_Station4.A_Remove(out => lrStation4Location);
				
			ELSE
				lrTargetLocation := lrStation3Location;
				Buffer_Station3.A_Remove(out => lrStation3Location);
				Buffer_Station4.A_Remove(out => lrStation4Location);
			
			END_IF
			iTableExecutor := 40;
			
		ELSIF Buffer_Station3.nCount = 0 AND Buffer_Station4.nCount = 0 THEN
			TableState := 0;//IDLE
			
		ELSE
			IF Buffer_Station3.nCount = 0 THEN
				lrTargetLocation := lrStation4Location;
				Buffer_Station4.A_Remove(out => lrStation4Location);
				
			ELSE
				lrTargetLocation := lrStation3Location;
				Buffer_Station3.A_Remove(out => lrStation3Location);
				
			END_IF
			iTableExecutor := 40;
		END_IF
		
//	21://get vision 3capture position
//		IF Vision3State = 0 THEN
//			Vision3State:= 10;
//			TableState:=22;
//		END_IF
//	22://get vision 4 capture position
//		IF Vision4State = 0 THEN
//			Vision4State:= 10;
//			TableState:=30;
//		END_IF
	
	40://MOVE POSITION
		fbRotaryTable.MR_MoveAbsolute(lrAbsolutePosition := lrTargetLocation);
		IF fbRotaryTable.InPosition THEN
			
			TableState := 41;
		END_IF
		
	41:// check position of vision station 3
		IF Vision3State = 0 THEN
			TableState := 42;
		END_IF
	42:
		Buffer_Station3.A_Get(out => lrCapPosStation3);
		bGetPictureStation3 := TRUE;
		
		IF LREAL_TO_INT(fbRotaryTable.ActualPosition) = LREAL_TO_INT(lrCapPosStation3) THEN
			Buffer_Station3.A_Remove(out => lrCapPosStation3);
			Vision3State:= 30;
			TableState := 43;
			
		ELSE
			bGetPictureStation3 := FALSE;
			TableState := 43;
			
		END_IF
			
	43:// check position of vision station 4
		IF Vision4State = 0 THEN
			TableState := 44;
		END_IF
	44:
		Buffer_Station4.A_Get(out => lrCapPosStation4);
		bGetPictureStation4 := TRUE;
		bResultProcessing := TRUE;
		
		IF LREAL_TO_INT(fbRotaryTable.ActualPosition) = LREAL_TO_INT(lrCapPosStation4) THEN
			Buffer_Station4.A_Remove(out => lrCapPosStation4);
			Vision4State:= 30;
			TableState := 60;
			
		ELSE
			bGetPictureStation4 := FALSE;
			bResultProcessing := FALSE;
			TableState := 60;
			
		END_IF
	
	
	
	
//	50://command vision 3
//		IF Vision3State = 0 THEN
//			Vision3State:= 20;
//			TableState:=55;
//		END_IF
//	55:	//command vision 4
//		IF Vision4State = 0 THEN
//			Vision4State:= 20;
//			TableState:=60;
//		END_IF

	
	
	
	
	60://check taking picture done
		IF NOT bGetPictureStation3 AND NOT bGetPictureStation4  AND NOT bResultProcessing THEN
			TableState := 70;
		END_IF
		
	70://state check result | product above table | buffer | go through sorting station
		IF bProductAboveTable THEN
			TableState := 10;//take product
		ELSIF Buffer_RotaryTable.nCount > 0 THEN
			TableState := 30;//get distance
		ELSE
			(* Make sure that the product is sorted *)
			fbRotaryTable.MR_MoveRelative(2*OneStep);
			IF fbRotaryTable.InPosition THEN
				
				TableState := 0;
			END_IF
			
		END_IF
	
END_CASE
///============================================================================================}}}
///(*==================================== Vision 3+4 process ====================================*){{{
CASE Vision3State OF
	0://idle | waiting
		;
//	10://get position in buffer
//		Buffer_Station3.A_Remove(out => lrCapPosStation3);
//		Vision3State := 0;

//	20://check position with table
//		bGetPictureStation3 := TRUE;
//		IF LREAL_TO_INT(fbRotaryTable.ActualPosition) = LREAL_TO_INT(lrCapPosStation3) THEN //convert from lreal to int for less precise
//			Vision3State:= 30;
//		ELSE
//			bGetPictureStation3 := FALSE;
//			Vision3State:= 0;
//		END_IF
			
	30://take picture cam 5+6
		IF doTriggerCam5.Command(PulseWidth:= T#1MS, DelayTimeForSecondTrigger:= T#34MS) AND
			doTriggerCam6.Command(PulseWidth:= T#1MS, DelayTimeForSecondTrigger:= T#34MS) THEN
			
			bGetPictureStation3 := FALSE;
			Vision3State := 0; 
		END_IF
		
END_CASE

(* station 4 have to take picture and request result from system *)
CASE Vision4State OF
	0:
		;
//	10://get trigger position in buffer
//		Buffer_Station4.A_Remove(out => lrCapPosStation4);
//		Vision4State := 0;

//	20://check trigger position with table position
//		bGetPictureStation4 := TRUE;
//		bResultProcessing 	:= TRUE;
//		IF LREAL_TO_INT(fbRotaryTable.ActualPosition) = LREAL_TO_INT(lrCapPosStation4) THEN //convert from lreal to int for less precise
//			Vision4State:= 30;
//		ELSE
//			bResultProcessing			:= FALSE;
//			bGetPictureStation4 		:= FALSE;
//			Vision4State:= 0;
//		END_IF
	
	30://trigger cam 7
		IF doTriggerCam7.Command(PulseWidth:= T#1MS, DelayTimeForSecondTrigger:= T#33MS) THEN
			bGetPictureStation4 := FALSE;
			Vision4State:= 40;
		END_IF
		
	40://request result
		(* testing purpose *)
		bResultGood:= TRUE;
		IF bResultGood THEN
			eFinalResult := VISION_RESULT_GOOD;
			bResultGood := FALSE;
			Vision4State:= 0;
		ELSIF bResultDirt THEN
			eFinalResult := VISION_RESULT_CONTAMINATION_DIRTY;
			bResultDirt := FALSE;
			Vision4State:= 0;
		ELSIF bResultDent THEN
			eFinalResult := VISION_RESULT_SCRATCH_DENT;
			bResultDent := FALSE;
			Vision4State:= 0;
		ELSIF bResultReject THEN
			eFinalResult := VISION_RESULT_REJECT;
			bResultReject := FALSE;
			Vision4State:= 0;
		END_IF

END_CASE
///============================================================================================}}}
///(*==================================== Sorting station ====================================*){{{
(* Add buffer for sorting station *)
CASE eFinalResult OF
	VISION_RESULT_UNKNOWN:
		;
	VISION_RESULT_GOOD:
		Buffer_SortGood.A_Add(in := fbRotaryTable.ActualPosition + lrSortGoodDistance);
		eFinalResult 		:= VISION_RESULT_UNKNOWN;
	VISION_RESULT_CONTAMINATION_DIRTY:
		Buffer_SortDirt.A_Add(in := fbRotaryTable.ActualPosition + lrSortDirtDistance);
		eFinalResult 		:= VISION_RESULT_UNKNOWN;
	VISION_RESULT_SCRATCH_DENT:
		Buffer_SortDent.A_Add(in := fbRotaryTable.ActualPosition + lrSortDentDistance);
		eFinalResult 		:= VISION_RESULT_UNKNOWN;
	VISION_RESULT_REJECT:
		Buffer_SortReject.A_Add(in := fbRotaryTable.ActualPosition + lrSortRejectDistance);
		eFinalResult 		:= VISION_RESULT_UNKNOWN;

END_CASE
(* Shoot the product out *)
(* Good case *)
CASE uSortGoodGetPosState OF
	0://idle | check buffer
		IF Buffer_SortGood.nCount > 0 THEN
			uSortGoodGetPosState:= 10;
		END_IF
	10://get position
		Buffer_SortGood.A_Get(out => lrSortGoodPos);
		uSortGoodGetPosState := 20;
	20://waiting table move in position | command table
		bResultProcessing 	:= FALSE;
		IF LREAL_TO_INT(fbRotaryTable.ActualPosition) <= LREAL_TO_INT(lrSortGoodPos) THEN
			uSortGoodGetPosState := 30;
		END_IF
	30://shoot it
		Buffer_SortGood.A_Remove(out => lrSortGoodPos);
		doBlowGood.Out := TRUE;
		uSortGoodGetPosState := 40;
		
	40://off
		tonGoodDelay(IN := TRUE, PT := tSortValveGoodTime);
		IF tonGoodDelay.Q THEN	
			doBlowGood.Out := FALSE;
			tonGoodDelay.IN := FALSE;
			uSortGoodGetPosState := 0;
		END_IF
		
END_CASE
(* DIRT CASE *)
CASE uSortDirtGetPosState OF
	0://idle | check buffer
		IF Buffer_SortDirt.nCount > 0 THEN
			uSortDirtGetPosState:= 10;
		END_IF
	10://get position
		Buffer_SortDirt.A_Get(out => lrSortDirtPos);
		uSortDirtGetPosState := 20;
	20://waiting table move in position | command table
		bResultProcessing 	:= FALSE;
		IF LREAL_TO_INT(fbRotaryTable.ActualPosition) <= LREAL_TO_INT(lrSortDirtPos) THEN
			uSortDirtGetPosState := 30;
		END_IF
	30://shoot it
		Buffer_SortDirt.A_Remove(out => lrSortDirtPos);
		doBlowDirtScratch.Out := TRUE;
		uSortDirtGetPosState := 40;
		
	40://off
		tonDirtDelay(IN := TRUE, PT := tSortValveDirtTime);
		IF tonDirtDelay.Q THEN	
			doBlowDirtScratch.Out := FALSE;
			tonDirtDelay.IN := FALSE;
			uSortDirtGetPosState := 0;
		END_IF
		
END_CASE
(* DENT CASE *)
CASE uSortDentGetPosState OF
	0://idle | check buffer
		IF Buffer_SortDent.nCount > 0 THEN
			uSortDentGetPosState:= 10;
		END_IF
	10://get position
		Buffer_SortDent.A_Get(out => lrSortDentPos);
		uSortDentGetPosState := 20;
	20://waiting table move in position | command table
		bResultProcessing 	:= FALSE;
		IF LREAL_TO_INT(fbRotaryTable.ActualPosition) <= LREAL_TO_INT(lrSortDentPos) THEN
			uSortDentGetPosState := 30;
		END_IF
	30://shoot it
		Buffer_SortDent.A_Remove(out => lrSortDentPos);
		doBlowDentContamination.Out := TRUE;
		uSortDentGetPosState := 40;
		
	40://off
		tonDentDelay(IN := TRUE, PT := tSortValveDentTime);
		IF tonDentDelay.Q THEN	
			doBlowDentContamination.Out := FALSE;
			tonDentDelay.IN := FALSE;
			uSortDentGetPosState := 0;
		END_IF
		
END_CASE
(* REJECT CASE *)
CASE uSortRejectGetPosState OF
	0://idle | check buffer
		IF Buffer_SortReject.nCount > 0 THEN
			uSortRejectGetPosState:= 10;
		END_IF
	10://get position
		Buffer_SortReject.A_Get(out => lrSortRejectPos);
		uSortRejectGetPosState := 20;
	20://waiting table move in position | command table
		bResultProcessing 	:= FALSE;
		IF LREAL_TO_INT(fbRotaryTable.ActualPosition) <= LREAL_TO_INT(lrSortRejectPos) THEN
			uSortRejectGetPosState := 30;
		END_IF
	30://shoot it
		Buffer_SortReject.A_Remove(out => lrSortRejectPos);
		doBlowReject.Out := TRUE;
		uSortRejectGetPosState := 40;
		
	40://off
		tonRejectDelay(IN := TRUE, PT := tSortValveRejectTime);
		IF tonRejectDelay.Q THEN	
			doBlowReject.Out := FALSE;
			tonRejectDelay.IN := FALSE;
			uSortRejectGetPosState := 0;
		END_IF
		
END_CASE
///============================================================================================}}}
(* control param *)
fbRobot.ref_CR800.Override:= 5;
uBufferTableCount:= Buffer_RotaryTable.nCount;

(* Mornitoring param *)
bActive 			:= fbRotaryTable.Active;
bBusy				:= fbRotaryTable.Busy;
bError 				:= fbRotaryTable.Error;
iErrorID 			:= fbRotaryTable.ErrorID;
iAxisErrorID 		:= fbRotaryTable.ErrorID;
lrActualPosition 	:= fbRotaryTable.ActualPosition;
rActualVelocity		:= fbRotaryTable.ActualVelocity;
bPowerOn 			:= fbRotaryTable.PowerOn;
bIsHomed 			:= fbRotaryTable.IsHomed;
bInVelocity			:= fbRotaryTable.InVelocity;
bInPostion 			:= fbRotaryTable.InPosition;
bMoveActive 		:= fbRotaryTable.MoveActive;
bJogDone 			:= fbRotaryTable.JogDone;
bStopped 			:= fbRotaryTable.Stopped;
bHalted 			:= fbRotaryTable.Halted;
eStatePlcOpen		:= fbRotaryTable.StatePlcOpen;

fbRobot.ref_CR800.Override:= 30;
fbRotaryTable.Velocity 			:= 50.0;
END_METHOD

END_FUNCTION_BLOCK

// ---- POUs/Machine/Module/Robot/FB_Robot.TcPOU
(*
Copyrights	: Operation Automation Department
Author		: HVAP
Description	: This function block is used to control robot and vision from RTC vendor
*)
FUNCTION_BLOCK FB_Robot IMPLEMENTS I_AOIRobot
VAR
	bFirstCycle 					: BOOL := TRUE;
	(* Auxilary *)
	tonDelay							: TON;		(* Provides any delay into the machine when switching something On/Off *)
	
	sName							: STRING;
	iOverride						: USINT;
	
	(* Properties *)
	_bActive						: BOOL;
	_bBusy							: BOOL;
	
	(* Components *)
	doRobotPowerOn					: FB_DigitalOutput;	(* Power on CR800 *)
	doRobotModeSwitch				: FB_DigitalOutput;	(* Set robot into automatic work mode *)
	
	(* Function blocks *)
	fbCR800 						: FB_CR800EtherCAT;
	
	(* CR800 EtherCAT diagnostic *)
	fbGetCR800EcState			:  FB_EcGetSlaveState;
	fbSetCR800CtrlState 		:  FB_EcReqSlaveState;		
	stCR800GetEcState			:  ST_EcSlaveState;		
	
	(* Robots EtherCAT communication *)
	sPLC_NET_ID 				: T_AmsNetId;// := '5.127.48.8.2.1'; //hardware config
	iCR800_1_ADDRESS			: UINT;//	:= 1003; //hardware config
	
	(* Action list *)
	eRobotAction				: E_AOIRobotActions;
	eRobotLastAction			: E_AOIRobotActions;
	
	(* State Machine *)
	eRobotState					: E_AOIRobotState;
	eRobotStateInit				: E_AOIRobotStateInit;
	eRobotStateAbort			: E_AOIRobotStateAbort;
	
END_VAR
(*
Version history:

+-------------+------------+----------------+----------+------------------------------------------+
|Date         | Version    | created under  | Author   | Remark                                   |
+=============+============+================+==========+==========================================+
|2024-02      | 1.0.0.0    | V3.1.4024.22   | HVAP     | Function block created                   |
+-------------+------------+----------------+----------+------------------------------------------+

*)

IF bFirstCycle THEN
	bFirstCycle := FALSE;
	fbCR800.MR_FirstCycle( sName := CONCAT(STR1 := sName, STR2 := ':CR800 Controler'), iOverride := iOverride);
	
	(* Assign digital output - robots power on switch *)
	doRobotPowerOn.MR_FirstCycle(	sName 		:= 'POWER ON',
									sModuleType := '',
									sPortID		:= '');
									
	(* Assign digital output - robots automatic mode switch *)
	doRobotModeSwitch.MR_FirstCycle(	sName 		:= 'MODE SWITCH',
										sModuleType := '',
										sPortID		:= '');
	
END_IF

_bActive := eRobotState >= E_AOIRobotState.READY_INITIALIZED;

(* Cyclic run *)
StateMachine();

fbCR800();

PROPERTY Active : BOOL
GET
Active := _bActive;
END_GET
END_PROPERTY

PROPERTY Busy : BOOL
GET
Busy := _bBusy;
END_GET
END_PROPERTY

METHOD M_EtherCATStatusCheck : BOOL
VAR_INST
	EtherCATStatusCheck : UINT;
END_VAR
CASE EtherCATStatusCheck OF
	
	0://MACHINE_STATE_UNINITIALIZED_CR800_ETHERCAT_STATUS_CHECK
		fbGetCR800EcState(			sNetId 		:= sPLC_NET_ID,
									nSlaveAddr	:= iCR800_1_ADDRESS,
									bExecute	:= TRUE,
									tTimeout 	:= DEFAULT_ADS_TIMEOUT,
									state		=> stCR800GetEcState);
		IF NOT fbGetCR800EcState.bBusy AND NOT fbGetCR800EcState.bError THEN
			fbGetCR800EcState(bExecute := FALSE);
			EtherCATStatusCheck := EtherCATStatusCheck + 10;
			
		END_IF
	
	10://MACHINE_STATE_UNINITIALIZED_CR800_ETHERCAT_STATUS_CHECK_DONE
		IF stCR800GetEcState.deviceState = EC_DEVICE_STATE_ERROR OR stCR800GetEcState.deviceState = 84 THEN
			EtherCATStatusCheck := 20;
			
		ELSIF stCR800GetEcState.deviceState = EC_DEVICE_STATE_SAFEOP THEN
			EtherCATStatusCheck := 30;
			
		ELSIF stCR800GetEcState.deviceState = EC_DEVICE_STATE_OP THEN
			EtherCATStatusCheck := 40;
		ELSE
			EtherCATStatusCheck := 0;
		END_IF
		
	20://MACHINE_STATE_UNINITIALIZED_CR800_ETHERCAT_ERROR_RESET
		fbSetCR800CtrlState( 		sNetId 		:= sPLC_NET_ID,
									nSlaveAddr	:= iCR800_1_ADDRESS,
									bExecute 	:= TRUE,
									tTimeout 	:= DEFAULT_ADS_TIMEOUT,
									state 		:= EC_DEVICE_STATE_ERROR);
		IF NOT fbSetCR800CtrlState.bBusy AND NOT fbSetCR800CtrlState.bError THEN
			fbSetCR800CtrlState(bExecute := FALSE);
			EtherCATStatusCheck := 0;
		END_IF
	
	30://MACHINE_STATE_UNINITIALIZED_CR800_ETHERCAT_REQUEST_OP_STATE
		fbSetCR800CtrlState( 		sNetId 		:= sPLC_NET_ID,
									nSlaveAddr	:= iCR800_1_ADDRESS,
									bExecute 	:= TRUE,
									tTimeout 	:= DEFAULT_ADS_TIMEOUT,
									state 		:= EC_DEVICE_STATE_OP);
		IF NOT fbSetCR800CtrlState.bBusy AND NOT fbSetCR800CtrlState.bError THEN
			fbSetCR800CtrlState(bExecute := FALSE);
			EtherCATStatusCheck := 0;
		END_IF

	40://MACHINE_STATE_UNINITIALIZED_CR800_CHECK_POWER_REGISTER
		IF fbCR800.CR800PoweredOn THEN
			EtherCATStatusCheck := 0;
			M_EtherCATStatusCheck := TRUE;
		END_IF
	
END_CASE
END_METHOD

METHOD M_PowerOnCommand : BOOL
VAR_INPUT
END_VAR
doRobotPowerOn.Out := TRUE;

tonDelay(IN := TRUE, PT := T#20S);
IF tonDelay.Q AND fbCR800.CR800PoweredOn THEN
	tonDelay(IN := FALSE);
	M_PowerOnCommand := TRUE;
END_IF
END_METHOD

PROPERTY ModeSwitch : BOOL
SET
doRobotModeSwitch.Out := ModeSwitch;
END_SET
END_PROPERTY

METHOD MR_Abort : BOOL
VAR_INPUT
END_VAR
IF eRobotState >= E_AOIRobotState.IDLE AND eRobotState <> E_AOIRobotState.ABORT  THEN
	_bBusy := TRUE;
	MR_Abort := FALSE;
	eRobotState := E_AOIRobotState.ABORT;
	eRobotStateAbort := E_AOIRobotStateAbort.CR800_RESET;
	
ELSIF eRobotState = E_AOIRobotState.UNINITIALIZED THEN
	_bBusy := FALSE;
	MR_Abort := TRUE;
	
END_IF
END_METHOD

METHOD MR_FirstCycle : BOOL
VAR_INPUT
	sName 				: STRING;
	iInitialOverride 	: USINT;
	sPLC_NET_ID			: T_AmsNetId;
	iCR800_1_ADDRESS	: UINT;
END_VAR
THIS^.sName := sName;
THIS^.iOverride := iInitialOverride;
THIS^.sPLC_NET_ID := sPLC_NET_ID;
THIS^.iCR800_1_ADDRESS := iCR800_1_ADDRESS;
END_METHOD

METHOD MR_GoBowl : BOOL
VAR_INPUT
END_VAR
IF eRobotState = E_AOIRobotState.IDLE THEN
	_bBusy := TRUE;
	MR_GoBowl := FALSE;
	eRobotState := E_AOIRobotState.GO_BOWL;
	
ELSIF eRobotState = E_AOIRobotState.ACTION_DONE THEN
	_bBusy := FALSE;
	MR_GoBowl := TRUE;
	
END_IF
END_METHOD

METHOD MR_GoHome : BOOL
VAR_INPUT
END_VAR
IF eRobotState = E_AOIRobotState.IDLE THEN
	_bBusy := TRUE;
	MR_GoHome := FALSE;
	eRobotState := E_AOIRobotState.GO_HOME;
	
ELSIF eRobotState = E_AOIRobotState.ACTION_DONE THEN
	_bBusy := FALSE;
	MR_GoHome := TRUE;
	
END_IF
END_METHOD

METHOD MR_GoInputProduct : BOOL
VAR_INPUT
END_VAR
IF eRobotState = E_AOIRobotState.IDLE THEN
	_bBusy := TRUE;
	MR_GoInputProduct := FALSE;
	eRobotState := E_AOIRobotState.GO_INPUT_PRODUCT;
	
ELSIF eRobotState = E_AOIRobotState.ACTION_DONE THEN
	_bBusy := FALSE;
	MR_GoInputProduct := TRUE;
	
END_IF
END_METHOD

METHOD MR_GoRotaryTable : BOOL
VAR_INPUT
END_VAR
IF eRobotState = E_AOIRobotState.IDLE THEN
	_bBusy := TRUE;
	MR_GoRotaryTable := FALSE;
	eRobotState := E_AOIRobotState.GO_ROTARY_TABLE;
	
ELSIF eRobotState = E_AOIRobotState.ACTION_DONE THEN
	_bBusy := FALSE;
	MR_GoRotaryTable := TRUE;
	
END_IF
END_METHOD

METHOD MR_GoStation1 : BOOL
VAR_INPUT
END_VAR
IF eRobotState = E_AOIRobotState.IDLE THEN
	_bBusy := TRUE;
	MR_GoStation1 := FALSE;
	eRobotState := E_AOIRobotState.GO_STATION_1;
	
ELSIF eRobotState = E_AOIRobotState.ACTION_DONE THEN
	_bBusy := FALSE;
	MR_GoStation1 := TRUE;
	
END_IF
END_METHOD

METHOD MR_GoStation2 : BOOL
VAR_INPUT
END_VAR
IF eRobotState = E_AOIRobotState.IDLE THEN
	_bBusy := TRUE;
	MR_GoStation2 := FALSE;
	eRobotState := E_AOIRobotState.GO_STATION_2;
	
ELSIF eRobotState = E_AOIRobotState.ACTION_DONE THEN
	_bBusy := FALSE;
	MR_GoStation2 := TRUE;
	
END_IF
END_METHOD

METHOD MR_Init : BOOL
VAR_INPUT
END_VAR
IF eRobotState = E_AOIRobotState.UNINITIALIZED THEN
	_bBusy := TRUE;
	MR_Init := FALSE;
	eRobotState := E_AOIRobotState.INITIALIZING;
	eRobotStateInit := E_AOIRobotStateInit.CR800_RESET;
	
ELSIF eRobotState = E_AOIRobotState.IDLE THEN
	_bBusy := FALSE;
	MR_Init := TRUE;
	
END_IF
END_METHOD

METHOD MR_Pick : BOOL
VAR_INPUT
END_VAR
IF eRobotState = E_AOIRobotState.IDLE THEN
	_bBusy := TRUE;
	MR_Pick := FALSE;
	eRobotState := E_AOIRobotState.PICK;
	
ELSIF eRobotState = E_AOIRobotState.ACTION_DONE THEN
	_bBusy := FALSE;
	MR_Pick := TRUE;
	
END_IF
END_METHOD

METHOD MR_Place : BOOL
VAR_INPUT
END_VAR
IF eRobotState = E_AOIRobotState.IDLE THEN
	_bBusy := TRUE;
	MR_Place := FALSE;
	eRobotState := E_AOIRobotState.PLACE;
	
ELSIF eRobotState = E_AOIRobotState.ACTION_DONE THEN
	_bBusy := FALSE;
	MR_Place := TRUE;
	
END_IF
END_METHOD

METHOD PROTECTED MS_Abort : BOOL
VAR_INPUT
END_VAR
CASE eRobotStateAbort OF
	E_AOIRobotStateAbort.CR800_RESET:
		fbCR800.MR_Reset();
		IF NOT fbCR800.Busy THEN
			eRobotStateAbort := E_AOIRobotStateAbort.CR800_ABORT;
		END_IF

	E_AOIRobotStateAbort.CR800_ABORT:
		fbCR800.MR_Abort();
		IF NOT fbCR800.Active THEN
			eRobotState := E_AOIRobotState.UNINITIALIZED;
		END_IF
		
END_CASE
END_METHOD

METHOD PROTECTED MS_ActionDone : BOOL
VAR_INPUT
END_VAR
IF NOT _bBusy THEN
	eRobotState := E_AOIRobotState.IDLE;
END_IF
END_METHOD

METHOD PROTECTED MS_GoBowl : BOOL
VAR_INPUT
END_VAR
fbCR800.ActionNumber := AOI_ROBOT_ACTION_GO_BOWL;
fbCR800.MR_DoAction(iActionNumber := fbCR800.ActionNumber);
IF NOT fbCR800.Busy THEN
	eRobotState := E_AOIRobotState.ACTION_DONE	;
END_IF
END_METHOD

METHOD PROTECTED MS_GoHome : BOOL
VAR_INPUT
END_VAR
fbCR800.MR_GoHome();
IF NOT fbCR800.Busy THEN
	eRobotState := E_AOIRobotState.ACTION_DONE;
END_IF
END_METHOD

METHOD PROTECTED MS_GoInputProduct : BOOL
VAR_INPUT
END_VAR
fbCR800.ActionNumber := AOI_ROBOT_ACTION_GO_INPUT_PRODUCT;
fbCR800.MR_DoAction(iActionNumber := fbCR800.ActionNumber);
IF NOT fbCR800.Busy THEN
	eRobotState := E_AOIRobotState.ACTION_DONE;
END_IF
END_METHOD

METHOD PROTECTED MS_GoRotaryTable : BOOL
VAR_INPUT
END_VAR
fbCR800.ActionNumber := AOI_ROBOT_ACTION_GO_TO_ROTARY_TABLE;
fbCR800.MR_DoAction(iActionNumber := fbCR800.ActionNumber);
IF NOT fbCR800.Busy THEN
	eRobotState := E_AOIRobotState.ACTION_DONE;
END_IF
END_METHOD

METHOD PROTECTED MS_GoStation1 : BOOL
VAR_INPUT
END_VAR
fbCR800.ActionNumber := AOI_ROBOT_ACTION_GO_TO_STATION_1;
fbCR800.MR_DoAction(iActionNumber := fbCR800.ActionNumber);
IF NOT fbCR800.Busy THEN
	eRobotState := E_AOIRobotState.ACTION_DONE;
END_IF
END_METHOD

METHOD PROTECTED MS_GoStation2 : BOOL
VAR_INPUT
END_VAR
fbCR800.ActionNumber := AOI_ROBOT_ACTION_GO_TO_STATION_2;
fbCR800.MR_DoAction(iActionNumber := fbCR800.ActionNumber);
IF NOT fbCR800.Busy THEN
	eRobotState := E_AOIRobotState.ACTION_DONE;
END_IF
END_METHOD

METHOD PROTECTED MS_Idle : BOOL
VAR_INPUT
END_VAR
;
END_METHOD

METHOD PROTECTED MS_Initializing : BOOL
VAR_INPUT
END_VAR
CASE eRobotStateInit OF
	E_AOIRobotStateInit.CR800_RESET:
		fbCR800.MR_Reset();
		IF NOT fbCR800.Busy THEN
			eRobotStateInit := E_AOIRobotStateInit.CR800_INIT;
		END_IF
	
	E_AOIRobotStateInit.CR800_INIT:
		fbCR800.MR_Init();
		IF fbCR800.Active THEN
			eRobotState := E_AOIRobotState.READY_INITIALIZED;
		END_IF
	
END_CASE
END_METHOD

METHOD PROTECTED MS_Pick : BOOL
VAR_INPUT
END_VAR
fbCR800.ActionNumber := AOI_ROBOT_ACTION_PICK;
fbCR800.MR_DoAction(iActionNumber := fbCR800.ActionNumber);
IF NOT fbCR800.Busy THEN
	eRobotState := E_AOIRobotState.ACTION_DONE;
END_IF
END_METHOD

METHOD PROTECTED MS_Place : BOOL
VAR_INPUT
END_VAR
fbCR800.ActionNumber := AOI_ROBOT_ACTION_PLACE;
fbCR800.MR_DoAction(iActionNumber := fbCR800.ActionNumber);
IF NOT fbCR800.Busy THEN
	eRobotState := E_AOIRobotState.ACTION_DONE;
END_IF
END_METHOD

METHOD PROTECTED MS_ReadyInitialized : BOOL
VAR_INPUT
END_VAR
eRobotState := E_AOIRobotState.IDLE;
END_METHOD

METHOD PROTECTED MS_Uninitialized : BOOL
VAR_INPUT
END_VAR
;
END_METHOD

PROPERTY ref_CR800 : REFERENCE TO FB_CR800EtherCAT
GET
ref_CR800 REF= fbCR800;
END_GET
END_PROPERTY

METHOD PROTECTED StateMachine : BOOL
VAR_INPUT
END_VAR
CASE eRobotState OF
	E_AOIRobotState.UNINITIALIZED:
		MS_Uninitialized();
		
	E_AOIRobotState.INITIALIZING:
		MS_Initializing();
		
	E_AOIRobotState.READY_INITIALIZED:
		MS_ReadyInitialized();
		
	E_AOIRobotState.IDLE:
		MS_Idle();

	E_AOIRobotState.PICK:
		MS_Pick();

	E_AOIRobotState.PLACE:
		MS_Place();

	E_AOIRobotState.GO_HOME:
		MS_GoHome();
		
	E_AOIRobotState.GO_BOWL:
		MS_GoBowl();
		
	E_AOIRobotState.GO_INPUT_PRODUCT:
		MS_GoInputProduct();
	
	E_AOIRobotState.GO_STATION_1:
		MS_GoStation1();
		
	E_AOIRobotState.GO_STATION_2:
		MS_GoStation2();
		
	E_AOIRobotState.GO_ROTARY_TABLE:	
		MS_GoRotaryTable();
		
	E_AOIRobotState.ACTION_DONE:
		MS_ActionDone();
		
	E_AOIRobotState.ABORT:
		MS_Abort();
		
END_CASE
END_METHOD

END_FUNCTION_BLOCK

// ---- POUs/Libs/Robots/Mitsubishi/FB_CR800EtherCAT.TcPOU
FUNCTION_BLOCK FB_CR800EtherCAT IMPLEMENTS I_CR800EtherCAT
VAR CONSTANT
	iMIN_ETHERCAT_REGISTER_IN_CR800	: INT 	:= 6000 ;	(*  *)
	iMAX_ETHERCAT_REGISTER_IN_CR800	: INT 	:= 6255 ;	(*  *)
	
	iSEND_REQUEST_ADDRESS			: UINT 	:= 6030 ;	(*  *)
	iRECEIVE_REQUEST_ADDRESS		: UINT 	:= 6031 ;	(*  *)
	
	tWATCHDOG_TIMEOUT				: TIME 	:= T#2S ;	(* Input timeout *)
END_VAR
VAR
	bFirstCycle			: BOOL := TRUE;	(* First cycle procedure bit *)
	sName				: STRING;		(*  *)
	
	stCR800EthercatData : ST_CR800EthercatData ;(* Data to map *)
	
	(* Internal commands *)
	bIsHomed					: BOOL;			(* Robot is it's home postion *)
	bReset						: BOOL;			(* Reset function block *)
	
	(* CR800 state *)
	bInit 						: BOOL;			(* Prepare a CR800 to work *)
	bGoHome 					: BOOL;			(* Moves a robot to the home postion *)
	bUpdateRecipes				: BOOL;			(* CR800 is updating recpies*)
	bGoAuto						: BOOL;			(* Robot goes to auto mode*)
	bDoAction					: BOOL;			(* Robot is doing action in automode*)
	bCycleStop					: BOOL;			(* Cr800 cycle is stopping *)
	bCyclePause					: BOOL;			(* Cr800 cycle is stopping *)
	bRestoreAuto				: BOOL;			(* CR800 is restoring auto mode *)
	bRestoreCycle				: BOOL;			(* CR800 is restoring cycle *)
	iActionNumber				: UINT;
	bAbort						: BOOL;			(* Deinitialize function block *)
	bError		 				: BOOL;			(* FB error occuring*)
	bDontSetInitialParameters	: BOOL;			(* Don't set initial parameters in initalization *)
	bBusy						: BOOL;
	bActive						: BOOL;
	bAutoModeStarted			: BOOL;
	bUninitialized				: BOOL; 
	bStopped					: BOOL;
	bInitProgram				: BOOL;
	bSendPosition1				: BOOL;
	bSendPosition2				: BOOL;
	bGetPosition				: BOOL;
	
	eErrorID 					: E_CR800Error;	(*  *)
	
	eCR800State					: E_CR800State					:= 0; (* Main state machine of function block *)
	eCR800StateBeforeReset		: E_CR800State					:= 0; (* State of CR800 before reseting the error *)
	eCR800StateHome 			: E_CR800StateHoming 			:= 0; (* State machine of homing *)
	eCR800StateDoRequest		: E_CR800StateDoingRequest		:= 0; (* State machine of executing request*)
	eCR800StateReceiveCommand	: E_CR800StateCommandExchange	:= 0; (* State machine of receive command data exchange *) 
	eCR800SendCommand			: E_CR800StateCommandExchange	:= 0; (* State machine of send commad data exchange *) 
	eCR800StateAbort 			: E_CR800StateAborting 			:= 0; (* State machine of aboriting *) 
	eCR800StateInitializing 	: E_CR800StateInitializing 		:= 0; (* State machine of initilaizing *)
	eCR800StateCycleStop 		: E_CR800StateCycleStopping		:= 0; (* State machine of cycle stopping *)
	eCR800StateCyclePause		: E_CR800StateCyclePausing		:= 0; (* State machine of cycle Pausing *)
	eCR800StateBeforeSendPosition : E_CR800State				:= 0;
	eCR800StateSendPosition		: E_CR800StateSendPosition		:= 0; (* State machine of cycle Pausing *)

	stRobot						: ST_VisuCtrlRobotFrame; 
	
	iOverride					: USINT;
	lrPositionX1				: LREAL;
	lrPositionY1				: LREAL;
	lrRotation1					: LREAL;
	lrPositionX2				: LREAL;
	lrPositionY2				: LREAL;
	lrRotation2					: LREAL;
	
	stUserDefinedArea			: ST_CR800UserDefinedArea;
	
	(* Timers *)
	tTimeout					: TIME := tWATCHDOG_TIMEOUT;	(**)
	tonWatchdog					: TON;							(* Input timeout watchdog *)

	feTrigStopped 				: F_TRIG;
	//rtErrorOccuring				: R_TRIG;
END_VAR

M_ConvertEthercatData() ;

//rtErrorOccuring(CLK := ErrorOccuring);
IF ErrorOccuring THEN
	//rtErrorOccuring(CLK := FALSE);
	eCR800State := CR800_IN_EXTERNAL_ERROR ;
	bError := TRUE ;
	eErrorID := CR800_ERROR_CR800_ERROR_OCCURING ;
END_IF

ActionNumber := iActionNumber;
stCR800EthercatData.arrRegistersOutput[6021] := USINT_TO_INT(iOverride);

StateMachine() ;

feTrigStopped(CLK := CycleStopping);

IF feTrigStopped.Q THEN 
	bStopped := TRUE;
END_IF

tonWatchdog(PT := tTimeout) ;

//stCR800EthercatData.arrRegistersOutput[6021] := 100 ; {warning 'Odhardkodować - przenieść do receptury'}

PROPERTY ActionNumber : UINT
GET
ActionNumber := iActionNumber;
END_GET
SET
IF ActionNumber >= 13 AND ActionNumber <= 100 THEN
	iActionNumber := ActionNumber;
END_IF
END_SET
END_PROPERTY

PROPERTY Active : REFERENCE TO BOOL
GET
Active REF= bActive;
END_GET
END_PROPERTY

PROPERTY AutoModeStarted : REFERENCE TO BOOL
GET
AutoModeStarted REF= bAutoModeStarted;
END_GET
END_PROPERTY

(* Desription from CR800 side:
"Outputs that the controller battery voltage is
low. The output is turned off when the
controller power supply is reconnected after
the battery replacement.
*The cumulative time where the controller
power supply is turned off exceeds 14600
hours.
The output is turned off if the battery depletion
time is reset." *)
{attribute 'monitoring' := 'variable'}
PROPERTY PUBLIC BatteryLow : BOOL ;
GET
BatteryLow := stCR800EthercatData.arrSignalsInputConverted[6014] ;
END_GET
END_PROPERTY

(* Desription from CR800 side:
Reset the battery cumulative tine. *) 
{attribute 'monitoring' := 'variable'}
PROPERTY BatteryReset : BOOL
GET
BatteryReset := stCR800EthercatData.arrSignalsOutputConverted[6015] ;
END_GET
SET
stCR800EthercatData.arrSignalsOutputConverted[6015] := BatteryReset ;
END_SET
END_PROPERTY

(* Desription from a CR800 side:
Output that the reset has been completed *)
{attribute 'monitoring' := 'variable'}
PROPERTY PUBLIC BatteryResetCompleted : BOOL ;
GET
BatteryResetCompleted := stCR800EthercatData.arrSignalsInputConverted[6015] ;
END_GET
END_PROPERTY

PROPERTY Busy : REFERENCE TO BOOL
GET
Busy REF= bBusy;
END_GET
END_PROPERTY

(* Desription from CR800 side:
Outputs that the power has been turned ON
and that the external input signal can be
received *)
{attribute 'monitoring' := 'variable'}
PROPERTY PUBLIC CR800PoweredOn : BOOL ;
GET
CR800PoweredOn := stCR800EthercatData.arrSignalsInputConverted[6000] ;
END_GET
END_PROPERTY

(* Desription from a CR800 side:
Starts the cycle stop *)
{attribute 'monitoring' := 'variable'}
PROPERTY CycleStop : BOOL
GET
CycleStop := stCR800EthercatData.arrSignalsOutputConverted[6013] ;
END_GET
SET
stCR800EthercatData.arrSignalsOutputConverted[6013] := CycleStop;
END_SET
END_PROPERTY

(* Desription from CR800 side:
"Outputs that the cycle stop is operating.
Turns OFF when the cycle stop is completed" *)
{attribute 'monitoring' := 'variable'}
PROPERTY PUBLIC CycleStopping : BOOL ;
GET
CycleStopping := stCR800EthercatData.arrSignalsInputConverted[6013] ;
END_GET
END_PROPERTY

PROPERTY DoingAction : REFERENCE TO BOOL
GET
DoingAction REF= bDoAction;
END_GET
END_PROPERTY

(*Desription from a CR800 side:
"Outputs that an emergency stop is occurring.
[EMGERR output conditions]
• External emergency stop error:
H0050, H0051 (Dual line is faulty)
• Operation panel emergency stop error:
H0060, H0061 (Dual line is faulty)
• T/B emergency stop error:
H0070, H0071 (Dual line is faulty)
• Door switch signal faulty:
H0039, H0040 (Dual line is faulty)
• Wiring error of EMG connector:
H0141"*)
{attribute 'monitoring' := 'variable'}
PROPERTY PUBLIC EmergencyStopOccuring : BOOL ;
GET
EmergencyStopOccuring := stCR800EthercatData.arrSignalsInputConverted[6016] ;
END_GET
END_PROPERTY

PROPERTY Error : REFERENCE TO BOOL
GET
Error REF= bError;
END_GET
END_PROPERTY

(* Actual FB error *)
{attribute 'monitoring' := 'variable'}
PROPERTY Errorname : STRING
GET
Errorname := TO_STRING(eErrorID) ;
END_GET
END_PROPERTY

{attribute 'monitoring' := 'variable'}
PROPERTY PUBLIC ErrorOccuring : BOOL ;
(*Desription from CR800 side:
Outputs that an error has occurred.
*)
GET
ErrorOccuring := stCR800EthercatData.arrSignalsInputConverted[6010] ;
END_GET
END_PROPERTY

(* Desription from CR800 side:
This input stops the program being executed.
(The specification is the same as for the STOP
parameter.)
Unlike the STOP parameter, signal numbers
can be changed. *)
{attribute 'monitoring' := 'variable'}
PROPERTY ErrorReset : BOOL
GET
ErrorReset := stCR800EthercatData.arrSignalsOutputConverted[6010] ;
END_GET
SET
stCR800EthercatData.arrSignalsOutputConverted[6010] := ErrorReset ;
END_SET
END_PROPERTY

PROPERTY EthercatData : REFERENCE TO ST_CR800EthercatData
GET
EthercatData REF= stCR800EthercatData;
END_GET
END_PROPERTY

(*Desription from CR800 side:
This output indicates that the controller mode
is set to AUTOMATIC.*)
{attribute 'monitoring' := 'variable'}
PROPERTY PUBLIC InAutomaticMode : BOOL ;
GET
InAutomaticMode := stCR800EthercatData.arrSignalsInputConverted[6003] ;
END_GET
END_PROPERTY

(* Desription from CR800 side:
This output indicates that the controller mode
is set to AUTOMATIC and remote operation
mode.*)
{attribute 'monitoring' := 'variable'}
PROPERTY PUBLIC InRemoteMode : BOOL ;
GET
InRemoteMode := stCR800EthercatData.arrSignalsInputConverted[6001] ;
END_GET
END_PROPERTY

(*Desription from CR800 side:
This output indicates that the controller mode
is set to Teaching mode. *)
{attribute 'monitoring' := 'variable'}
PROPERTY PUBLIC InTeachingMode : BOOL ;
GET
InTeachingMode := stCR800EthercatData.arrSignalsInputConverted[6002] ;
END_GET
END_PROPERTY

PROPERTY IsHomed : REFERENCE TO BOOL
GET
IsHomed REF= bIsHomed;
END_GET
END_PROPERTY

(*This mehtod converts raw data from memory and converts its number for the same like in the mitshubishi manual
  F:\Dept\SMT\Electronics\Mitsubishi\Manuals\Karta ethercat*)
METHOD Protected M_ConvertEthercatData : BOOL
VAR
	iLoop	: INT;	
END_VAR
FOR iLoop := 0 TO 31 DO  
	stCR800EthercatData.arrSignalsInputConverted[iMIN_ETHERCAT_REGISTER_IN_CR800  +iLoop*8]	:= 	stCR800EthercatData.arrSignalsInputRaw[iLoop].0	;
	stCR800EthercatData.arrSignalsInputConverted[iMIN_ETHERCAT_REGISTER_IN_CR800+1+iLoop*8]	:= 	stCR800EthercatData.arrSignalsInputRaw[iLoop].1	;
	stCR800EthercatData.arrSignalsInputConverted[iMIN_ETHERCAT_REGISTER_IN_CR800+2+iLoop*8] := 	stCR800EthercatData.arrSignalsInputRaw[iLoop].2	;
	stCR800EthercatData.arrSignalsInputConverted[iMIN_ETHERCAT_REGISTER_IN_CR800+3+iLoop*8] := 	stCR800EthercatData.arrSignalsInputRaw[iLoop].3	;
	stCR800EthercatData.arrSignalsInputConverted[iMIN_ETHERCAT_REGISTER_IN_CR800+4+iLoop*8] := 	stCR800EthercatData.arrSignalsInputRaw[iLoop].4	;
	stCR800EthercatData.arrSignalsInputConverted[iMIN_ETHERCAT_REGISTER_IN_CR800+5+iLoop*8] := 	stCR800EthercatData.arrSignalsInputRaw[iLoop].5	;
	stCR800EthercatData.arrSignalsInputConverted[iMIN_ETHERCAT_REGISTER_IN_CR800+6+iLoop*8] := 	stCR800EthercatData.arrSignalsInputRaw[iLoop].6	;
	stCR800EthercatData.arrSignalsInputConverted[iMIN_ETHERCAT_REGISTER_IN_CR800+7+iLoop*8] := 	stCR800EthercatData.arrSignalsInputRaw[iLoop].7	;
	
	stCR800EthercatData.arrSignalsOutputRaw[iLoop].0	:=	stCR800EthercatData.arrSignalsOutputConverted[iMIN_ETHERCAT_REGISTER_IN_CR800  +iLoop*8];
	stCR800EthercatData.arrSignalsOutputRaw[iLoop].1	:=	stCR800EthercatData.arrSignalsOutputConverted[iMIN_ETHERCAT_REGISTER_IN_CR800+1+iLoop*8];
	stCR800EthercatData.arrSignalsOutputRaw[iLoop].2	:=	stCR800EthercatData.arrSignalsOutputConverted[iMIN_ETHERCAT_REGISTER_IN_CR800+2+iLoop*8];
	stCR800EthercatData.arrSignalsOutputRaw[iLoop].3	:=	stCR800EthercatData.arrSignalsOutputConverted[iMIN_ETHERCAT_REGISTER_IN_CR800+3+iLoop*8];
	stCR800EthercatData.arrSignalsOutputRaw[iLoop].4	:=	stCR800EthercatData.arrSignalsOutputConverted[iMIN_ETHERCAT_REGISTER_IN_CR800+4+iLoop*8];
	stCR800EthercatData.arrSignalsOutputRaw[iLoop].5	:=	stCR800EthercatData.arrSignalsOutputConverted[iMIN_ETHERCAT_REGISTER_IN_CR800+5+iLoop*8];
	stCR800EthercatData.arrSignalsOutputRaw[iLoop].6	:=	stCR800EthercatData.arrSignalsOutputConverted[iMIN_ETHERCAT_REGISTER_IN_CR800+6+iLoop*8];
	stCR800EthercatData.arrSignalsOutputRaw[iLoop].7	:=	stCR800EthercatData.arrSignalsOutputConverted[iMIN_ETHERCAT_REGISTER_IN_CR800+7+iLoop*8];
END_FOR
END_METHOD

(* 1 - Request executed, 0 - request not executed 
	Description:
		This method doing request robot to do request with given number in iNumberOfRequest *)

METHOD PROTECTED M_DoRequest : BOOL
VAR_INPUT
	iNumberOfRequest	: 	UINT	;	(* Destination memory place in the robot*)
END_VAR
CASE eCR800StateDoRequest OF

	CR800_DOING_REQUEST_IDLE:
		M_DoRequest			:= FALSE ;
		eCR800StateDoRequest		:= CR800_DOING_REQUEST_SEND_REQUEST;
		
	CR800_DOING_REQUEST_SEND_REQUEST:
		IF M_SendCommand(iDestinationAdress := iSEND_REQUEST_ADDRESS, iRequestNumber := iNumberOfRequest) THEN
			eCR800StateDoRequest	:= CR800_DOING_REQUEST_WAIT_FOR_CONFIRM;
		END_IF
		
	CR800_DOING_REQUEST_WAIT_FOR_CONFIRM:
		IF M_ReceiveCommand(iDestinationAdress := iRECEIVE_REQUEST_ADDRESS) THEN
			eCR800StateDoRequest 	:= CR800_DOING_REQUEST_DONE ;
		END_IF
	
	CR800_DOING_REQUEST_DONE:
		M_DoRequest			:= TRUE ;
		eCR800StateDoRequest 		:= CR800_DOING_REQUEST_IDLE ;
END_CASE
END_METHOD

(*1 - Operation rights granted, 0 - Operation rights not granted
	Description: 
		This method grants operation rights to the PLC in CR800
		IE. PLC is only controlling the robot.
		Warning: The operation rights is lost, when teaching box is in the "Operation panel" screen.
		Input bRequest: 1 - Enable, 0 - unable *) 

METHOD PROTECTED M_OperationRigtsEnable : BOOL 
VAR_INPUT
	bRequest : BOOL ; (*1 - Enable, 0 - unable *) 
END_VAR
IF bRequest THEN 
	OperationRightsEnable := TRUE ;
	tonWatchdog.IN := TRUE ;
	IF OperationRightsEnabled THEN
		tonWatchdog.IN := FALSE ;
		M_OperationRigtsEnable := TRUE ;
	//ELSIF tonWatchdog.Q THEN
	//	bError 		:= TRUE ;
	//	eErrorID	:= CR800_ERROR_GRANTING_OPERATION_RIGHTS_TIMED_OUT ;			
	END_IF
END_IF

IF NOT bRequest THEN 
	OperationRightsEnable := FALSE ;
	tonWatchdog.IN := TRUE ;
	IF NOT OperationRightsEnabled THEN
		tonWatchdog.IN := FALSE ;
		M_OperationRigtsEnable := FALSE ;
	ELSIF tonWatchdog.Q THEN
		bError 		:= TRUE ;
		eErrorID	:= CR800_ERROR_ABORTING_OPERATION_RIGHTS_TIMED_OUT ;			
	END_IF
END_IF
END_METHOD

(* 1 - Program is reseted, 0 - program is not reseted
	Description:
		This method reset the program in Cr800
		IE. The next program start will begin form the first line*)
METHOD PROTECTED M_ProgramReset : BOOL
VAR_INPUT
END_VAR
IF ProgramOperating THEN
	bError 		:= TRUE ;
	eErrorID	:= CR800_ERROR_CANT_RESET_PRG_DURING_PRG_RUN ;
ELSE
	ProgramReset 	:= TRUE	;
	tonWatchdog.IN 	:= TRUE ;
	IF ProgramSelectionEnabled THEN
		ProgramReset 	:= FALSE;
		tonWatchdog.IN 	:= FALSE;	
		M_ProgramReset := TRUE ;
	ELSIF tonWatchdog.Q THEN
		bError 			:= TRUE ;
		eErrorID		:= CR800_ERROR_RESET_PRG_TIMED_OUT ;			
	END_IF
END_IF
END_METHOD

(* 0 - program not started, 1 - Program started 
	Description:
		This method starts the program in CR800 *) 
METHOD protected M_ProgramStart : BOOL
IF tonWatchdog.Q THEN
	bError 			:= TRUE ;
	eErrorID		:= CR800_ERROR_START_PRG_TIMED_OUT ;	
ELSIF NOT ProgramOperating OR StopSTS THEN
	ProgramStart 	:= TRUE	;
	M_ProgramStart := FALSE;
	tonWatchdog.IN 	:= TRUE ;
ELSIF ProgramOperating THEN
	ProgramStart 	:= FALSE;
	M_ProgramStart := TRUE ;
	tonWatchdog.IN 	:= FALSE;		
END_IF
END_METHOD

(* 1 - program stopped, 0 - program has not stopped
	Description:
		This method stops (pause) the program in CR800.
		IE. Stops the program implicitly *)
METHOD PROTECTED  M_ProgramStop : BOOL
M_ProgramStop  := FALSE ;
ProgramStop2 	:= TRUE ;

IF StopSTS AND NOT ProgramOperating THEN
	ProgramStop2	:= FALSE ;
	M_ProgramStop  := TRUE ;
END_IF
END_METHOD

(* 0 - command not Received, 1 - command Received 
	Desription:
		This method waits for the information from the iDestinationAddress, send confirmation,
 		waits for reset command and then resets confirmation *)
{attribute 'monitoring' := 'variable'}
METHOD PROTECTED M_ReceiveCommand : BOOL 
VAR_INPUT
	iDestinationAdress	: 	UINT	;	(* Destination memory place in the robot*)
END_VAR
//IF tonWatchdog.Q THEN
//	bError 		:= TRUE ;
//	eErrorID	:= CR800_ERROR_RECEIVE_COMMAND_TIMED_OUT ;			
//END_IF

CASE eCR800StateReceiveCommand OF
	
	CR800_CMD_EXCHANGE_IDLE:
		M_ReceiveCommand := FALSE ;
//		tonWatchdog.IN 	:= TRUE ;
		eCR800StateReceiveCommand 	:= CR800_CMD_EXCHANGE_WAIT_FOR_DATA ;

	CR800_CMD_EXCHANGE_WAIT_FOR_DATA:
		IF stCR800EthercatData.arrSignalsInputConverted[iDestinationAdress] THEN
			eCR800StateReceiveCommand := CR800_CMD_EXCHANGE_SEND_CONFIRMATION ;			
		END_IF

	CR800_CMD_EXCHANGE_SEND_CONFIRMATION:
		stCR800EthercatData.arrSignalsOutputConverted[iDestinationAdress] := TRUE ;
		eCR800StateReceiveCommand 	:= CR800_CMD_EXCHANGE_WAIT_FOR_RESET_COMMAND ;
		
	CR800_CMD_EXCHANGE_WAIT_FOR_RESET_COMMAND:
		IF NOT stCR800EthercatData.arrSignalsInputConverted[iDestinationAdress] THEN
			eCR800StateReceiveCommand := CR800_CMD_EXCHANGE_RESET_ITERLOCKS ;			
		END_IF
			
	CR800_CMD_EXCHANGE_RESET_ITERLOCKS:
		stCR800EthercatData.arrSignalsOutputConverted[iDestinationAdress] := FALSE;
		eCR800StateReceiveCommand	:= CR800_CMD_EXCHANGE_DONE ;

	CR800_CMD_EXCHANGE_DONE:
//		tonWatchdog.IN 					:= FALSE;	
		M_ReceiveCommand 				:= TRUE ;		
		eCR800StateReceiveCommand	:= CR800_CMD_EXCHANGE_IDLE ;

END_CASE
END_METHOD

(* Desription:
	This method resets fb variables *)
METHOD PROTECTED M_ResetVariables : BOOL
VAR
	iLoop: INT;
END_VAR
//M_OperationRigtsEnable(bRequest 	:= 0);
eCR800StateDoRequest				:= 0 ;
eCR800StateHome 					:= 0 ;	
eCR800StateReceiveCommand			:= 0 ;
eCR800SendCommand					:= 0 ;
eCR800StateInitializing 			:= 0 ;
eCR800StateCycleStop 				:= 0 ; 
eCR800StateCyclePause				:= 0 ; 
eCR800StateSendPosition				:= 0 ;

eErrorID := CR800_ERROR_OK;

bGoHome 			:=	FALSE;
bUpdateRecipes		:=	FALSE;
bGoAuto				:=	FALSE;
bDoAction			:=	FALSE;
bCycleStop			:=	FALSE;
bCyclePause			:= 	FALSE;
bRestoreCycle		:=  FALSE;
bIsHomed			:=	FALSE;
bAutoModeStarted 	:=  FALSE;
tonWatchdog.IN 		:=  FALSE;

FOR iLoop := iMIN_ETHERCAT_REGISTER_IN_CR800 TO iMAX_ETHERCAT_REGISTER_IN_CR800 DO
	stCR800EthercatData.arrRegistersOutput[iLoop] 			:= 0 ;
	stCR800EthercatData.arrSignalsOutputConverted[iLoop]	:= 0 ;
END_FOR
END_METHOD

(* 0 - command not sent, 1 - command sent 
	Descritpion:
		This method sends the information to the iDestinationAddress, waits for a confirmation,
 		send reset command and then resets send request *)
{attribute 'monitoring' := 'variable'}
METHOD PROTECTED M_SendCommand : BOOL

VAR_INPUT
	iDestinationAdress		: 	UINT	;	(* Destination memory place in the robot*)
	iRequestNumber			:  	UINT	;	(* Reqest number that robot has to perform *)		
END_VAR
IF tonWatchdog.Q THEN
	bError 		:= TRUE ;
	eErrorID	:= CR800_ERROR_SEND_COMMAND_TIMED_OUT ;			
END_IF


CASE eCR800SendCommand OF
	
	CR800_CMD_EXCHANGE_IDLE:
		M_SendCommand 	:= FALSE ;
		RequestNumber 	:= iRequestNumber ; 
		tonWatchdog.IN 	:= TRUE ;
		eCR800SendCommand 	:= CR800_CMD_EXCHANGE_SEND_DATA ;

	CR800_CMD_EXCHANGE_SEND_DATA:
		stCR800EthercatData.arrSignalsOutputConverted[iDestinationAdress] := TRUE ;
		eCR800SendCommand 	:= CR800_CMD_EXCHANGE_WAIT_FOR_CONFIRMATION ;
		
	CR800_CMD_EXCHANGE_WAIT_FOR_CONFIRMATION:
		IF stCR800EthercatData.arrSignalsInputConverted[iDestinationAdress] THEN
			eCR800SendCommand := CR800_CMD_EXCHANGE_RESET_ITERLOCKS ;			
		END_IF
	
	CR800_CMD_EXCHANGE_RESET_ITERLOCKS:
		stCR800EthercatData.arrSignalsOutputConverted[iDestinationAdress] := FALSE;
		eCR800SendCommand	:= CR800_CMD_EXCHANGE_WAIT_FOR_RESET_CONFIRMATION ;
	
	CR800_CMD_EXCHANGE_WAIT_FOR_RESET_CONFIRMATION:
		IF NOT stCR800EthercatData.arrSignalsInputConverted[iDestinationAdress] THEN
			eCR800SendCommand := CR800_CMD_EXCHANGE_DONE ;			
		END_IF
		
	CR800_CMD_EXCHANGE_DONE:
		tonWatchdog.IN 				:= FALSE;
		M_SendCommand 				:= TRUE ;
		eCR800SendCommand 	:= CR800_CMD_EXCHANGE_IDLE ;
END_CASE
END_METHOD

(* Servo Off request. 1 - Servo offed succesfully, 0 - Servo has not stopped yet
	Description:
		This method turns off the servos of the robot *)
METHOD PROTECTED M_ServoOff : BOOL
ServoOFF := TRUE ;

IF ServoIsOff THEN
	ServoOFF 	:= FALSE ;
	M_ServoOFF := TRUE ;
END_IF
END_METHOD

(* 1 - Servo on succesfully, 0 - Servo has not stopped yet
	Description:
		This method turns on the servos of the robot *)
METHOD PROTECTED M_ServoOn : BOOL (*Servo ON request*)
IF NOT ServoOFF THEN

	ServoON 		:= TRUE ;
	tonWatchdog.IN 	:= TRUE ;
	IF ServoIsOn THEN
		ServoON 		:= FALSE ;
		M_ServoON 		:= TRUE	 ;
		tonWatchdog.IN 	:= FALSE ;
	ELSIF tonWatchdog.Q THEN
		bError 		:= TRUE ;
		eErrorID	:= CR800_ERROR_SERVO_ON_TIMED_OUT ;			
	END_IF
	
END_IF
END_METHOD

(* Actual state of main state machine *)
{attribute 'monitoring' := 'variable'}
PROPERTY MainStateMachine : STRING
GET
MainStateMachine := TO_STRING(eCR800State) ;
END_GET
END_PROPERTY

(* 1 - abroting finished, 0 - aborting not finished.
	Description:
		This method aborts all actions, stops and reset the program and turn off the robot*)
METHOD  MR_Abort : BOOL
IF eCR800State <> CR800_UNINITIALIZED OR ServoIsOn THEN
	bBusy 	:= TRUE;
	bAbort := TRUE;
	MR_Abort := FALSE;
	eCR800State := CR800_ABORTING;
	fbMachineLogger.MR_AddLogs(CONCAT(sName,' : abort requested'));	
	
ELSIF eCR800State = CR800_UNINITIALIZED THEN
	bAbort := FALSE;
	MR_Abort := TRUE;
//	bActive := FALSE; 
	bBusy 	:= FALSE;
	fbMachineLogger.MR_AddLogs(CONCAT(sName,' : abort done'));	
	
END_IF
END_METHOD

(* 1 - During reseting, 0 - Reset completed
	Description:
		Reset the batetery replacement timer request.
		Indirectly resets the battery error. *) 
METHOD MR_BatteryReset : BOOL
IF NOT BatteryResetCompleted THEN
	bBusy 	:= TRUE;
	MR_BatteryReset := TRUE;
	BatteryReset :=	TRUE;
	fbMachineLogger.MR_AddLogs(CONCAT(sName,' : battery reset requested'));
	
ELSE 
	MR_BatteryReset := FALSE;
	BatteryReset :=	FALSE;
	bBusy 	:= FALSE;
	fbMachineLogger.MR_AddLogs(CONCAT(sName,' : battery reset done'));
	
END_IF
END_METHOD

(* 1 - Cycle paused, 0 - Cycle not paused
	Description:
		This method stop the program without reseting.
		IE. stops movement implicily 
		To restore the movement use MR_RestoreCycle or MR_GoHome *)
METHOD MR_CyclePause : BOOL
IF eCR800State = CR800_DOING_ACTION THEN
	bBusy 	:= TRUE;
	bCyclePause := TRUE;
	MR_CyclePause := FALSE;
	eCR800State := E_CR800State.CR800_CYCLE_PAUSING;
	fbMachineLogger.MR_AddLogs(CONCAT(sName,' : cycle pausing requested'));
	
ELSIF eCR800State = E_CR800State.CR800_CYCLE_PAUSING_DONE THEN
	bCyclePause	:= FALSE;
	MR_CyclePause := TRUE;
	bBusy 	:= FALSE;
	fbMachineLogger.MR_AddLogs(CONCAT(sName,' : cycle pausing done'));
	
END_IF
END_METHOD

(* 1 - During stopping, 0 - Cycle stop completed
	Description:
		This method stop the program, when the "End" command is met in the robots program.
		Caution: It stops the program AND reset it. To restore it you need to use MR_RestoreAuto. *) 

METHOD MR_CycleStop : BOOL
IF eCR800State = CR800_DOING_ACTION OR eCR800State = CR800_IDLE_CYCLE_PAUSED OR eCR800State = CR800_IDLE_AUTO_PAUSED THEN
	bBusy 	:= TRUE;
	bCycleStop 	:= TRUE;
	MR_CycleStop := FALSE;
	eCR800State := CR800_CYCLE_STOPPING;
	fbMachineLogger.MR_AddLogs(CONCAT(sName,' : cycle stopping requested'));
	
ELSIF eCR800State = CR800_CYCLE_STOPING_DONE THEN
	bDoAction := FALSE;
	bCycleStop := FALSE;
	MR_CycleStop := TRUE;
	bBusy 	:= FALSE;
	fbMachineLogger.MR_AddLogs(CONCAT(sName,' : cycle stopping done'));
	
END_IF
END_METHOD

(* 0 - Action not completed, 1 - Action completed
Description:
This method send request to do an action.
Robot will perform an action number that is called in input.
If the action is single and has and end use:
	IF MR_DoAction( iActionNumber := iExampleNumber) THEN
		bDO_A_FLIP := true ;
	END_IF
If the action is endless then just call it, and then use MR_CycleStop.
	MR_DoAction( iActionNumber := iExampleNumber) *)
METHOD MR_DoAction : BOOL
VAR_INPUT
	iActionNumber : UINT ;
END_VAR
IF eCR800State = CR800_IDLE_AUTO THEN
	IF iActionNumber <= 12 THEN 
		bError := TRUE ;
		eErrorID := CR800_ERROR_CANT_DO_SYSTEM_ACTION_IN_THIS_REQUEST ;
	ELSE
		bBusy 	:= TRUE;
		bDoAction := TRUE;
		bStopped := FALSE;
		MR_DoAction := FALSE;
		iActionNumber := iActionNumber;
		eCR800State := CR800_DOING_ACTION;
		fbMachineLogger.MR_AddLogs(FUN_MergeStrings5(sName,' : doing action number: ',UINT_TO_STRING(iActionNumber), '',' requested'));
	
	END_IF
	
ELSIF eCR800State = CR800_DOING_ACTION_DONE THEN
	bIsHomed := FALSE;
	bAutoModeStarted := FALSE;
	MR_DoAction := TRUE;
	bBusy := FALSE; 
	fbMachineLogger.MR_AddLogs(FUN_MergeStrings5(sName,' : doing action number: ',UINT_TO_STRING(iActionNumber),'',' done'));
	
ELSIF eCR800State <> CR800_DOING_ACTION AND eCR800State = E_CR800State.CR800_IDLE_CYCLE_PAUSED 
	AND eCR800State <> E_CR800State.CR800_CYCLE_PAUSING AND eCR800State <> E_CR800State.CR800_CYCLE_PAUSING
	AND eCR800State <> CR800_CYCLE_RESTORING AND eCR800State <> CR800_CYCLE_RESTORING_DONE THEN
	bError := TRUE ;
	eErrorID := CR800_ERROR_CANT_DO_ACTION_WITHOUT_BEEING_AUTO ;
	fbMachineLogger.MR_AddLogs(CONCAT(sName,' : ERROR_CANT_DO_ACTION_WITHOUT_BEEING_AUTO'));
	
END_IF
END_METHOD

METHOD MR_FirstCycle : BOOL
VAR_INPUT
	sName 				: STRING;
	iOverride			: USINT;
END_VAR
THIS^.sName := sName;
THIS^.iOverride := iOverride;
END_METHOD

(* 0 - FB is NOT in auto mode, 1 - FB is in auto mode
	Description:
		This method reqest FB to go into the auto mode. In automode FB can perform actions (MR_DoAction) *)
METHOD MR_GoAuto : BOOL
IF NOT bIsHomed THEN 
	bError := TRUE ;
	eErrorID := CR800_ERROR_CANT_GO_AUTO_WITHOUT_BEEING_HOMED ;
	fbMachineLogger.MR_AddLogs(CONCAT(sName,' : ERROR_CANT_GO_AUTO_WITHOUT_BEEING_HOMED'));
	
ELSIF eCR800State = CR800_IDLE_HOMED OR eCR800State = CR800_IDLE_CYCLE_PAUSED THEN
	bBusy 	:= TRUE;
	bGoAuto := TRUE;
	MR_GoAuto := FALSE;
	iActionNumber := stRobot.iActionNumber;
	eCR800State := CR800_GOING_AUTO;
	fbMachineLogger.MR_AddLogs(CONCAT(sName,' : going auto requested'));
	
ELSIF eCR800State = CR800_GOING_AUTO_DONE THEN
	bStopped := FALSE;
	bGoAuto := FALSE;
	MR_GoAuto := TRUE;
	bAutoModeStarted := TRUE;
	bBusy 	:= FALSE;
	fbMachineLogger.MR_AddLogs(CONCAT(sName,' : going auto done'));
	
END_IF
END_METHOD

(* 1 - Homing finished, 0 - Homing not finished.
	Description:
	This method request the robot to go home *)
METHOD MR_GoHome : BOOL
IF eCR800State = CR800_IDLE_NOT_HOMED OR eCR800State = CR800_IDLE_AUTO OR eCR800State = CR800_IDLE_AUTO_PAUSED THEN
	bBusy 	:= TRUE;	
	bGoHome := TRUE;
	MR_GoHome := FALSE;
	eCR800State := CR800_GOING_HOME;
	fbMachineLogger.MR_AddLogs(CONCAT(sName,' : going home requested'));
	
ELSIF eCR800State = CR800_GOING_HOME_DONE THEN
	bIsHomed := TRUE;
	bGoHome := FALSE;
	MR_GoHome := TRUE;
	bBusy 	:= FALSE;
	fbMachineLogger.MR_AddLogs(CONCAT(sName,' : going home done'));
	
END_IF
END_METHOD

(* 1 - Initializing finished, 0 - Initializing not finished.
	Description:
		This method initialize the robot:
			1. Checks for ethercat connection
			2. Checks for power of the CR800
			3. Checks for emergency stop
			4. Checks is CR800 is in auto mode
			5. Enable rights
			6. Turn on servos
			7. Resets the program
			8. Starts the program
			9. Sets initial parameters in the robot (when initializing after error this step is ommited) *)
METHOD MR_Init : BOOL
IF eCR800State = CR800_UNINITIALIZED AND NOT bAbort AND NOT bReset THEN
	bBusy 	:= TRUE;
	bInit := TRUE;
	MR_Init := FALSE;
	eCR800State := CR800_INITIALIZING;
	fbMachineLogger.MR_AddLogs(CONCAT(sName,' : initialization requested'));
	
ELSIF eCR800State = CR800_READY_INITIALIZED THEN
	bUninitialized := FALSE;
	bActive := TRUE;
	bInit := FALSE;
	MR_Init := TRUE;
	bBusy 	:= FALSE;
	fbMachineLogger.MR_AddLogs(CONCAT(sName,' : initialization done'));
	
END_IF
END_METHOD

(* 1 - Reset finished, 0 - Reset not finished.
	Description:
		This method resets the error state of the FB *)
METHOD MR_Reset : BOOL
IF eCR800State < CR800_RESET AND bError THEN
	bBusy 	:= TRUE;
	bReset := TRUE;
	eCR800StateBeforeReset := eCR800State;
	MR_Reset := FALSE;
	eCR800State := CR800_RESET;
	fbMachineLogger.MR_AddLogs(CONCAT(sName,' : reset requested'));
	
ELSIF eCR800State = CR800_RESET_DONE THEN
	bReset := FALSE;
	MR_Reset := TRUE;
	bBusy 	:= FALSE;
	fbMachineLogger.MR_AddLogs(CONCAT(sName,' : reset done'));
		
END_IF
END_METHOD

(* 1 - Reset finished, 0 - Reset not finished.
	Description:
		This method resets the internal error of CR800 *)
METHOD MR_ResetCR800Err : BOOL
IF ErrorOccuring  THEN
	bBusy 	:= TRUE;
	MR_ResetCR800Err := FALSE;
	ErrorReset := TRUE;
	fbMachineLogger.MR_AddLogs(CONCAT(sName,' : controller reset requested'));
	
ELSE 
	ErrorReset := FALSE;
	MR_ResetCR800Err := TRUE;	
	bBusy 	:= FALSE;
	fbMachineLogger.MR_AddLogs(CONCAT(sName,' : controller reset done'));
	
END_IF
END_METHOD

(* 1 - Auto mode restored, 0 - Auto mode NOT restored.
	Description:
		This method restores auto mode after the MR_CycleStop method *)
METHOD MR_RestoreAuto : BOOL
IF eCR800State = CR800_IDLE_AUTO_PAUSED THEN
	bBusy 	:= TRUE;
	bRestoreAuto := TRUE;
	bInitProgram := TRUE;
	MR_RestoreAuto := FALSE;
	eCR800State := CR800_AUTO_RESTORING;
	fbMachineLogger.MR_AddLogs(CONCAT(sName,' : restoring auto mode requested'));
	
ELSIF eCR800State = CR800_AUTO_RESTORING_DONE THEN
	bStopped := FALSE;
	bRestoreAuto := FALSE;
	bInitProgram := FALSE;
	MR_RestoreAuto := TRUE;
	bBusy 	:= FALSE;
	fbMachineLogger.MR_AddLogs(CONCAT(sName,' : restoring auto mode done'));
	
END_IF
END_METHOD

(* 1 - Cycle restored, 0 - Cycle NOT restored.
	Description:
		This method restores cycle after the MR_CyclePause method *)
METHOD MR_RestoreCycle : BOOL

VAR
	FA: BOOL;
END_VAR
IF eCR800State = CR800_IDLE_CYCLE_PAUSED THEN
	bBusy 	:= TRUE;
	bRestoreCycle := TRUE;
	MR_RestoreCycle	:= FALSE;
	eCR800State := CR800_CYCLE_RESTORING;
	fbMachineLogger.MR_AddLogs(CONCAT(sName,' : restoring cycle requested'));
		
ELSIF eCR800State = CR800_CYCLE_RESTORING_DONE THEN	
	bRestoreCycle := FALSE;
	MR_RestoreCycle := TRUE;
	bBusy 	:= FALSE;
	fbMachineLogger.MR_AddLogs(CONCAT(sName,' : restoring cycle done'));
	
END_IF
END_METHOD

METHOD MR_SendPosition1 : BOOL 
VAR_INPUT
	lrPositionX1	: LREAL;
	lrPositionY1	: LREAL;
	lrRotation1		: LREAL;
END_VAR
IF eCR800State = CR800_DOING_ACTION OR eCR800State = CR800_IDLE_AUTO_PAUSED OR eCR800State = CR800_IDLE_AUTO OR eCR800State = CR800_IDLE_HOMED OR eCR800State = CR800_IDLE_NOT_HOMED THEN
	bBusy 	:= TRUE;
	bSendPosition1 := TRUE;
	MR_SendPosition1 := FALSE;
	eCR800StateBeforeSendPosition := eCR800State;
	eCR800State := CR800_SEND_POSITION_1;
	eCR800StateSendPosition := CR800_SEND_POSITION_CONVERTING;
	THIS^.lrPositionX1 := lrPositionX1;
	THIS^.lrPositionY1 := lrPositionY1;
	THIS^.lrRotation1 := lrRotation1;
	fbMachineLogger.MR_AddLogs(CONCAT(sName,' : sending first position requested'));
	
ELSIF eCR800State = CR800_SEND_POSITION_1_DONE THEN
	bSendPosition1	:= FALSE;
	MR_SendPosition1 := TRUE;
	//bBusy := FALSE;
	fbMachineLogger.MR_AddLogs(CONCAT(sName,' : sending first position done'));
	
END_IF
END_METHOD

METHOD MR_SendPosition2 : BOOL 
VAR_INPUT
	lrPositionX2	: LREAL;
	lrPositionY2	: LREAL;
	lrRotation2		: LREAL;
END_VAR
IF eCR800State = CR800_DOING_ACTION OR eCR800State = CR800_IDLE_AUTO_PAUSED OR eCR800State = CR800_IDLE_AUTO OR eCR800State = CR800_IDLE_HOMED OR eCR800State = CR800_IDLE_NOT_HOMED THEN
	bBusy 	:= TRUE;
	bSendPosition2 := TRUE;
	MR_SendPosition2 := FALSE;
	eCR800StateBeforeSendPosition := eCR800State;
	eCR800State := CR800_SEND_POSITION_2;
	eCR800StateSendPosition := CR800_SEND_POSITION_CONVERTING;
	THIS^.lrPositionX2 := lrPositionX2;
	THIS^.lrPositionY2 := lrPositionY2;
	THIS^.lrRotation2 := lrRotation2;
	fbMachineLogger.MR_AddLogs(CONCAT(sName,' : sending second position requested'));
	
ELSIF eCR800State = CR800_SEND_POSITION_2_DONE THEN
	bSendPosition2	:= FALSE;
	MR_SendPosition2 := TRUE;
	//bBusy := FALSE;
	fbMachineLogger.MR_AddLogs(CONCAT(sName,' : sending second position done'));
	
END_IF
END_METHOD

(* 1 - Recipies updated, 0 - Recipies not updated.
	Description:
		This method updated the recipies, while robot is homed *)
METHOD MR_UpdateRecipies : BOOL
IF eCR800State = CR800_IDLE_HOMED THEN
	bBusy 	:= TRUE;
	bUpdateRecipes := TRUE;
	MR_UpdateRecipies := FALSE;
	eCR800State := CR800_UPDATING_RECIPIES;
	fbMachineLogger.MR_AddLogs(CONCAT(sName,' : updating recipes requested'));
	
ELSIF eCR800State = CR800_UPDATE_RECIPIES_DONE THEN
	bUpdateRecipes := FALSE;
	MR_UpdateRecipies := TRUE;
	bBusy 	:= FALSE;
	fbMachineLogger.MR_AddLogs(CONCAT(sName,' : updating recipes done'));
	
END_IF
END_METHOD

METHOD PROTECTED  MS_Aborting
CASE eCR800StateAbort OF
	
	CR800_ABORTING_IDLE:
		eCR800StateAbort := CR800_ABORTING_ENABLE_RIGHTS;
	
	CR800_ABORTING_ENABLE_RIGHTS:
		IF M_OperationRigtsEnable(bRequest := TRUE) THEN
			eCR800StateAbort := CR800_ABORTING_PRGM_STOP;
		END_IF
	
	CR800_ABORTING_PRGM_STOP: 
		IF M_ProgramStop() THEN
			eCR800StateAbort := CR800_ABORTING_PRGM_RESET ;
		END_IF
	
	CR800_ABORTING_PRGM_RESET: 
		IF M_ProgramReset() THEN
			IF NOT bInitProgram THEN
				eCR800StateAbort := CR800_ABORTING_SERVO_OFF ;
			ELSE 
				eCR800StateAbort := CR800_ABORTING_DONE ;
			END_IF
		END_IF
		
	CR800_ABORTING_SERVO_OFF: 
		IF M_ServoOFF() THEN
			eCR800StateAbort := CR800_ABORTING_DONE ;
		END_IF
	 
	CR800_ABORTING_DONE:
	
		M_OperationRigtsEnable(bRequest 	:= 0);
		eCR800StateDoRequest				:= 0 ;
		eCR800StateHome 					:= 0 ;	
		eCR800StateReceiveCommand			:= 0 ;
		eCR800SendCommand					:= 0 ;
		eCR800StateInitializing 			:= 0 ;
		eCR800StateCycleStop 				:= 0 ; 
		eCR800StateCyclePause				:= 0 ; 
		bGoHome 			:=	FALSE;
		bUpdateRecipes		:=	FALSE;
		bGoAuto				:=	FALSE;
		bDoAction			:=	FALSE;
		bCycleStop			:=	FALSE;
		bCyclePause			:= 	FALSE;
		bRestoreCycle		:=  FALSE;
		bIsHomed			:=	FALSE;
		bAutoModeStarted 	:=  FALSE;
		tonWatchdog.IN 		:=  FALSE;
		bInit				:= 	FALSE;
		
		IF NOT bInitProgram THEN
			eCR800State := CR800_UNINITIALIZED;
		ELSE 
			eCR800State := CR800_INITIALIZING;
		END_IF	
			
		eCR800StateAbort := CR800_ABORTING_IDLE ;
END_CASE
END_METHOD

METHOD PROTECTED MS_CyclePauseDone
IF NOT bCyclePause THEN
	eCR800State := CR800_IDLE_CYCLE_PAUSED ;
END_IF
END_METHOD

METHOD PROTECTED MS_CyclePausing
CASE eCR800StateCyclePause OF
	CR800_CYCLE_PAUSING_IDLE:
		eCR800StateCyclePause := E_CR800StateCyclePausing.CR800_CYCLE_PAUSING;
		
	E_CR800StateCyclePausing.CR800_CYCLE_PAUSING:
		IF M_ProgramStop() THEN
			eCR800StateCyclePause := E_CR800StateCyclePausing.CR800_CYCLE_PAUSING_DONE;
		END_IF
		
	E_CR800StateCyclePausing.CR800_CYCLE_PAUSING_DONE:
		eCR800State := E_CR800State.CR800_CYCLE_PAUSING_DONE;
		eCR800StateCyclePause := CR800_CYCLE_PAUSING_IDLE;
END_CASE
END_METHOD

METHOD PROTECTED MS_CycleStopDone
IF NOT bCycleStop THEN
	eCR800State := CR800_IDLE_AUTO_PAUSED ;
END_IF
END_METHOD

METHOD PROTECTED MS_CycleStopping
VAR_INST
	tonWait : TON := (pt := T#1S) ;
END_VAR
CASE eCR800StateCycleStop OF
	CR800_CYCLE_STOPPPING_IDLE:
		eCR800StateCycleStop := CR800_CYCLE_STOPPPING_SEND_REQUEST;
		
	CR800_CYCLE_STOPPPING_SEND_REQUEST:
		CycleStop := TRUE ;
		eCR800StateCycleStop := CR800_CYCLE_STOPPPING_WAIT_FOR_STOP;

	CR800_CYCLE_STOPPPING_WAIT_FOR_STOP:
		tonWait.IN := TRUE ;
		IF NOT CycleStopping AND tonWait.Q THEN
			eCR800StateCycleStop := CR800_CYCLE_STOPPPING_RESET_VARIABLES;
		END_IF
		
	CR800_CYCLE_STOPPPING_RESET_VARIABLES:
		tonWait.IN := FALSE ;
		bDoAction := FALSE;
		eCR800StateReceiveCommand := 0;
		eCR800SendCommand := 0;
		eCR800StateDoRequest := 0; 	
		eCR800StateCycleStop := CR800_CYCLE_STOPPPING_DONE;
		
	CR800_CYCLE_STOPPPING_DONE:
		CycleStop := FALSE ;
		eCR800State := CR800_CYCLE_STOPING_DONE;
		eCR800StateCycleStop := CR800_CYCLE_STOPPPING_IDLE ;
END_CASE

tonWait();
END_METHOD

METHOD PROTECTED MS_DoAction_Done
bDoAction := FALSE;
eCR800State := CR800_IDLE_AUTO ;
END_METHOD

METHOD PROTECTED MS_DoingAction
IF M_DoRequest(iNumberOfRequest := iActionNumber) THEN
	eCR800State := CR800_DOING_ACTION_DONE ;
END_IF
END_METHOD

METHOD PROTECTED MS_GoAutoDone
IF NOT bGoAuto THEN
	eCR800State := CR800_IDLE_AUTO ;
END_IF
END_METHOD

METHOD PROTECTED MS_GoHomeDone
IF NOT bGoHome THEN
	eCR800State := CR800_IDLE_HOMED ;
END_IF
END_METHOD

METHOD PROTECTED MS_GoingAuto
IF M_DoRequest(E_RobotSystemActions.GO_AUTO) THEN
	eCR800State := CR800_GOING_AUTO_DONE ;
END_IF
END_METHOD

METHOD PROTECTED MS_GoingHome
CASE eCR800StateHome OF

	CR800_HOMING_IDLE:
		IF eCR800State = CR800_IDLE_AUTO OR eCR800State = CR800_IDLE_AUTO_PAUSED THEN
			eCR800StateHome	:= CR800_HOMING_RESET_PROGRAM ;
		ELSE 
			eCR800StateHome	:= CR800_HOMING_SEND_REQUEST ;
		END_IF
		
	CR800_HOMING_RESET_PROGRAM:
		IF M_ProgramReset() THEN
			eCR800StateHome := CR800_HOMING_RESET_CYCLE_VARIABLES ;
		END_IF	
		
	CR800_HOMING_RESET_CYCLE_VARIABLES:
		bDoAction := FALSE;
		eCR800StateReceiveCommand := 0;
		eCR800SendCommand := 0;
		eCR800StateDoRequest := 0;
		eCR800StateHome := CR800_HOMING_START_PROGRAM ;	
	
		
	CR800_HOMING_START_PROGRAM:
		IF M_ProgramStart() THEN
			eCR800StateHome := CR800_HOMING_SEND_REQUEST ;
		END_IF
	
	CR800_HOMING_SEND_REQUEST:
		IF M_DoRequest(E_RobotSystemActions.DO_HOMING) THEN   
			eCR800StateHome := CR800_HOMING_DONE ;
		END_IF	
		
	CR800_HOMING_DONE:
		eCR800State := CR800_GOING_HOME_DONE ;
		eCR800StateHome := CR800_HOMING_IDLE ;
END_CASE
END_METHOD

METHOD PROTECTED MS_IdleAuto
;
END_METHOD

METHOD PROTECTED MS_IdleAutoPaused
;
END_METHOD

METHOD PROTECTED MS_IdleCyclePaused
;
END_METHOD

METHOD PROTECTED MS_IdleHomed
;
END_METHOD

METHOD PROTECTED MS_IdleNotHomed
;
END_METHOD

METHOD PROTECTED MS_InExternalError
bDontSetInitialParameters := TRUE;
END_METHOD

METHOD PROTECTED MS_Initializing
CASE eCR800StateInitializing OF
		
	CR800_INIT_IDLE:
		eCR800StateInitializing := CR800_INIT_ETHERCAT_CHCEK ;
		
	CR800_INIT_ETHERCAT_CHCEK:
		tonWatchdog.IN := TRUE ;
		IF stCR800EthercatData.iInfoDataState = 8 THEN
			tonWatchdog.IN := FALSE ;	
			eCR800StateInitializing := CR800_INIT_POWER_CHCECK;
		ELSIF tonWatchdog.Q THEN
			bError := TRUE ;
			eErrorID := CR800_ERROR_ETHERCAT_CHECK_FAIL ;			
		END_IF
	
	CR800_INIT_POWER_CHCECK:
		tonWatchdog.IN := TRUE ;
		IF CR800PoweredOn THEN
			tonWatchdog.IN := FALSE ;	
			eCR800StateInitializing := CR800_INIT_EMERG_STOP_CHCECK;
		ELSIF tonWatchdog.Q THEN
			bError := TRUE ;
			eErrorID := CR800_ERROR_POWER_CHECK_FAIL ;			
		END_IF
		
		
	CR800_INIT_EMERG_STOP_CHCECK:
		tonWatchdog.IN := TRUE ;
		IF NOT EmergencyStopOccuring THEN
			tonWatchdog.IN := FALSE ;	
			eCR800StateInitializing := CR800_INIT_CHECK_FOR_AUTO_MODE;
		ELSIF tonWatchdog.Q THEN
			bError := TRUE ;
			eErrorID := CR800_ERROR_EMERGENCY_STOP_OCCURING ;			
		END_IF
		
	CR800_INIT_CHECK_FOR_AUTO_MODE:
		tonWatchdog.IN := TRUE;
		IF InAutomaticMode THEN
			tonWatchdog.IN 			:= FALSE ;	
			eCR800StateInitializing := CR800_INIT_ENABLE_RIGHTS;
		ELSIF tonWatchdog.Q THEN
			bError := TRUE ;
			eErrorID := CR800_ERROR_AUTO_MODE_CHECK_FAIL ;		
		END_IF
		
	CR800_INIT_ENABLE_RIGHTS:
		IF M_OperationRigtsEnable(bRequest := TRUE) THEN
			eCR800StateInitializing	:= CR800_INIT_SERVO_ON ;
		END_IF
		
	CR800_INIT_SERVO_ON:
		IF M_ServoON() THEN
			eCR800StateInitializing	:= CR800_INIT_PROGRAM_RESET ;
		END_IF
		
	CR800_INIT_PROGRAM_RESET:
		IF M_ProgramReset() THEN
			eCR800StateInitializing	:= CR800_INIT_PROGRAM_START ;
		END_IF
			
	CR800_INIT_PROGRAM_START:
		IF M_ProgramStart() THEN
			IF bDontSetInitialParameters THEN 
				bDontSetInitialParameters := FALSE ;
				eCR800StateInitializing := CR800_INIT_DONE ;			
			ELSE
				eCR800StateInitializing := CR800_INIT_SET_INITIAL_PARAMETERS_REQUEST ;				
			END_IF
		END_IF	

	CR800_INIT_SET_INITIAL_PARAMETERS_REQUEST: 
		IF M_DoRequest(iNumberOfRequest := E_RobotSystemActions.SET_INITIAL_PARAMETERS) THEN
			eCR800StateInitializing := CR800_INIT_DONE ;
		END_IF

	CR800_INIT_DONE:
		IF NOT bInitProgram THEN
			eCR800State := CR800_READY_INITIALIZED;
		ELSE
			eCR800State := CR800_AUTO_RESTORING_DONE;
		END_IF
		eCR800StateInitializing := CR800_INIT_IDLE ;
			
END_CASE
END_METHOD

METHOD PROTECTED MS_ReadyInitialized
VAR_INPUT
END_VAR
eCR800State := CR800_IDLE_NOT_HOMED;
END_METHOD

METHOD PROTECTED MS_Reset
VAR_INPUT
END_VAR
M_ResetVariables();
IF MR_ResetCR800Err() THEN
	eCR800State := CR800_RESET_DONE;
	eErrorID := CR800_ERROR_OK;
	bError := FALSE;
END_IF
END_METHOD

METHOD PROTECTED MS_ResetDone
VAR_INPUT
END_VAR
IF NOT bReset THEN
	IF eCR800StateBeforeReset >= CR800_IDLE_NOT_HOMED  THEN
		eCR800State := CR800_IDLE_NOT_HOMED ;
	ELSE
		eCR800State := CR800_UNINITIALIZED ;
	END_IF
END_IF
END_METHOD

METHOD PROTECTED MS_RestoreAutoDone
IF NOT bRestoreAuto THEN
	eCR800State := CR800_IDLE_NOT_HOMED ;
END_IF
END_METHOD

METHOD PROTECTED MS_RestoreCycleDone
IF NOT bRestoreCycle THEN
	eCR800State := CR800_DOING_ACTION ;
END_IF
END_METHOD

METHOD PROTECTED MS_RestoringAuto
eCR800State := CR800_ABORTING ;
END_METHOD

METHOD PROTECTED MS_RestoringCycle
IF M_ProgramStart() THEN 
	eCR800State := CR800_CYCLE_RESTORING_DONE ;
END_IF
END_METHOD

METHOD PROTECTED MS_SendingPosition1
VAR_INST
	lrPositionXFirstHalf  	: LREAL;
	lrPositionXSecondHalf  	: LREAL;
	lrPositionYFirstHalf  	: LREAL;
	lrPositionYSecondHalf 	: LREAL;
	lrRotationFirstHalf  	: LREAL;
	lrRotationSecondHalf	: LREAL;
END_VAR
CASE eCR800StateSendPosition OF 
	CR800_SEND_POSITION_CONVERTING:
		LTRUNC( lr_in := lrPositionX1,
				LTRUNC => lrPositionXFirstHalf);
		LTRUNC( lr_in := lrPositionY1,
				LTRUNC => lrPositionYFirstHalf);
		LTRUNC( lr_in := lrRotation1,
				LTRUNC => lrRotationFirstHalf);
	
		FRAC( lr_in := lrPositionX1,
				FRAC => lrPositionXSecondHalf);
		FRAC( lr_in := lrPositionY1,
				FRAC => lrPositionYSecondHalf);
		FRAC( lr_in := lrRotation1,
				FRAC => lrRotationSecondHalf);
				
		eCR800StateSendPosition := CR800_SEND_POSITION_SENDING;
		
	CR800_SEND_POSITION_SENDING:
		stCR800EthercatData.arrRegistersOutput[6022] :=	LREAL_TO_INT(lrPositionXFirstHalf); 
		stCR800EthercatData.arrRegistersOutput[6023] :=	LREAL_TO_INT(1000 * lrPositionXSecondHalf); 
		stCR800EthercatData.arrRegistersOutput[6024] :=	LREAL_TO_INT(lrPositionYFirstHalf); 
		stCR800EthercatData.arrRegistersOutput[6025] :=	LREAL_TO_INT(1000 * lrPositionYSecondHalf); 
		stCR800EthercatData.arrRegistersOutput[6026] :=	LREAL_TO_INT(lrRotationFirstHalf); 
		stCR800EthercatData.arrRegistersOutput[6027] :=	LREAL_TO_INT(1000 * lrRotationSecondHalf); 
			
		eCR800State := CR800_SEND_POSITION_1_DONE;
		
END_CASE
END_METHOD

METHOD PROTECTED MS_SendingPosition1Done
IF NOT bSendPosition1 THEN
	eCR800State := eCR800StateBeforeSendPosition;
	bBusy := FALSE;
	
END_IF
END_METHOD

